LIN {X 0,Y 288.913,Z 1256.965,A -85,B 0,C 180,E1 22492.445,E2 22492.445} C_VEL
LIN {X 0,Y 288.678,Z 1266.037,A -85,B 0,C 180,E1 22499.979,E2 22499.979} C_VEL
LIN {X 0,Y 289.252,Z 1269.357,A -85,B 0,C 180,E1 22505.992,E2 22505.992} C_VEL
LIN {X 0,Y 291.406,Z 1269.606,A -85,B 0,C 180,E1 22511.982,E2 22511.982} C_VEL
LIN {X 0,Y 298.511,Z 1264.594,A -85,B 0,C 180,E1 22520.789,E2 22520.789} C_VEL
LIN {X 0,Y 311.662,Z 1253.252,A -85,B 0,C 180,E1 22529.064,E2 22529.064} C_VEL
LIN {X 0,Y 331.336,Z 1236.016,A -85,B 0,C 180,E1 22536.45,E2 22536.45} C_VEL
LIN {X 0,Y 358.772,Z 1211.951,A -85,B 0,C 180,E1 22542.947,E2 22542.947} C_VEL
LIN {X 0,Y 361.993,Z 1209.216,A -85,B 0,C 180,E1 22543.83,E2 22543.83} C_VEL
LIN {X 0,Y 333.812,Z 1237.362,A -85,B 0,C 180,E1 22549.712,E2 22549.712} C_VEL
LIN {X 0,Y 313.92,Z 1258.852,A -85,B 0,C 180,E1 22556.298,E2 22556.298} C_VEL
LIN {X 0,Y 299.966,Z 1275.518,A -85,B 0,C 180,E1 22563.783,E2 22563.783} C_VEL
LIN {X 0,Y 291.853,Z 1286.905,A -85,B 0,C 180,E1 22571.864,E2 22571.864} C_VEL
LIN {X 0,Y 289.278,Z 1291.684,A -85,B 0,C 180,E1 22577.92,E2 22577.92} C_VEL
LIN {X 0,Y 288.568,Z 1293.172,A -85,B 0,C 180,E1 22585.704,E2 22585.704} C_VEL
LIN {X 0,Y 288.992,Z 1290.468,A -85,B 0,C 180,E1 22591.516,E2 22591.516} C_VEL
LIN {X 0,Y 289.159,Z 1283.794,A -85,B 0,C 180,E1 22597.542,E2 22597.542} C_VEL
LIN {X 0,Y 290.047,Z 1270.937,A -85,B 0,C 180,E1 22604.382,E2 22604.382} C_VEL
LIN {X 0,Y 290.956,Z 1264.711,A -85,B 0,C 180,E1 22607.439,E2 22607.439} C_VEL
LIN {X 0,Y 296.193,Z 1251.831,A -85,B 0,C 180,E1 22614.979,E2 22614.979} C_VEL
LIN {X 0,Y 306.956,Z 1232.131,A -85,B 0,C 180,E1 22622.484,E2 22622.484} C_VEL
LIN {X 0,Y 322.234,Z 1206.9,A -85,B 0,C 180,E1 22628.957,E2 22628.957} C_VEL
LIN {X 0,Y 340.074,Z 1177.254,A -85,B 0,C 180,E1 22634.139,E2 22634.139} C_VEL
LIN {X 0,Y 358.674,Z 1143.561,A -85,B 0,C 180,E1 22638.141,E2 22638.141} C_VEL
LIN {X 0,Y 372.662,Z 1114.646,A -85,B 0,C 180,E1 22640.6,E2 22640.6} C_VEL
LIN {X 0,Y 373.421,Z 1108.193,A -85,B 0,C 180,E1 22642.533,E2 22642.533} C_VEL
LIN {X 0,Y 372.674,Z 1104.982,A -85,B 0,C 180,E1 22645.328,E2 22645.328} C_VEL
LIN {X 0,Y 372.153,Z 1105.867,A -85,B 0,C 180,E1 22648.785,E2 22648.785} C_VEL
LIN {X 0,Y 371.792,Z 1111.104,A -85,B 0,C 180,E1 22651.662,E2 22651.662} C_VEL
LIN {X 0,Y 356.868,Z 1141.073,A -85,B 0,C 180,E1 22654.392,E2 22654.392} C_VEL
LIN {X 0,Y 341.823,Z 1166.001,A -85,B 0,C 180,E1 22657.887,E2 22657.887} C_VEL
LIN {X 0,Y 327.191,Z 1186.173,A -85,B 0,C 180,E1 22662.219,E2 22662.219} C_VEL
LIN {X 0,Y 325.799,Z 1187.915,A -85,B 0,C 180,E1 22662.7,E2 22662.7} C_VEL
LIN {X 0,Y 316.07,Z 1196.775,A -85,B 0,C 180,E1 22664.784,E2 22664.784} C_VEL
LIN {X 0,Y 307.469,Z 1203.336,A -85,B 0,C 180,E1 22666.77,E2 22666.77} C_VEL
LIN {X 0,Y 306.628,Z 1204.067,A -85,B 0,C 180,E1 22667.118,E2 22667.118} C_VEL
LIN {X 0,Y 296.611,Z 1212.121,A -85,B 0,C 180,E1 22672.684,E2 22672.684} C_VEL
LIN {X 0,Y 291.006,Z 1214.857,A -85,B 0,C 180,E1 22677.037,E2 22677.037} C_VEL
LIN {X 0,Y 285.807,Z 1214.307,A -85,B 0,C 180,E1 22683.06,E2 22683.06} C_VEL
LIN {X 0,Y 283.385,Z 1208.666,A -85,B 0,C 180,E1 22689.252,E2 22689.252} C_VEL
LIN {X 0,Y 283.421,Z 1196.875,A -85,B 0,C 180,E1 22695.723,E2 22695.723} C_VEL
LIN {X 0,Y 285.142,Z 1180.307,A -85,B 0,C 180,E1 22701.438,E2 22701.438} C_VEL
LIN {X 0,Y 288.35,Z 1157.172,A -85,B 0,C 180,E1 22706.829,E2 22706.829} C_VEL
LIN {X 0,Y 292.258,Z 1130.682,A -85,B 0,C 180,E1 22711.033,E2 22711.033} C_VEL
LIN {X 0,Y 296.178,Z 1100.104,A -85,B 0,C 180,E1 22714.268,E2 22714.268} C_VEL
LIN {X 0,Y 299.485,Z 1062.201,A -85,B 0,C 180,E1 22716.707,E2 22716.707} C_VEL
LIN {X 0,Y 298.982,Z 1051.383,A -85,B 0,C 180,E1 22717.371,E2 22717.371} C_VEL
LIN {X 0,Y 282.969,Z 995.061,A -85,B 0,C 180,E1 22721.869,E2 22721.869} C_VEL
LIN {X 0,Y 277.408,Z 977.53,A -85,B 0,C 180,E1 22723.544,E2 22723.544} C_VEL
LIN {X 0,Y 277.257,Z 977.53,A -85,B 0,C 180,E1 22733.028,E2 22733.028} C_VEL
LIN {X 0,Y 277.681,Z 977.53,A -85,B 0,C 180,E1 22740.854,E2 22740.854} C_VEL
LIN {X 0,Y 278.202,Z 977.53,A -85,B 0,C 180,E1 22747.851,E2 22747.851} C_VEL
LIN {X 0,Y 278.682,Z 977.53,A -85,B 0,C 180,E1 22754.21,E2 22754.21} C_VEL
LIN {X 0,Y 279.215,Z 977.53,A -85,B 0,C 180,E1 22760.616,E2 22760.616} C_VEL
LIN {X 0,Y 279.937,Z 977.53,A -85,B 0,C 180,E1 22766.883,E2 22766.883} C_VEL
LIN {X 0,Y 279.933,Z 977.53,A -85,B 0,C 180,E1 22773.088,E2 22773.088} C_VEL
LIN {X 0,Y 278.942,Z 977.53,A -85,B 0,C 180,E1 22782.535,E2 22782.535} C_VEL
LIN {X 0,Y 278.361,Z 977.53,A -85,B 0,C 180,E1 22789.048,E2 22789.048} C_VEL
LIN {X 0,Y 277.861,Z 977.53,A -85,B 0,C 180,E1 22795.85,E2 22795.85} C_VEL
LIN {X 0,Y 277.467,Z 977.53,A -85,B 0,C 180,E1 22804.97,E2 22804.97} C_VEL
LIN {X 0,Y 277.579,Z 977.96,A -85,B 0,C 180,E1 22805.92,E2 22805.92} C_VEL
LIN {X 0,Y 300.397,Z 1034.729,A -85,B 0,C 180,E1 22811.695,E2 22811.695} C_VEL
LIN {X 0,Y 313.014,Z 1073.998,A -85,B 0,C 180,E1 22815.793,E2 22815.793} C_VEL
LIN {X 0,Y 317.958,Z 1093.026,A -85,B 0,C 180,E1 22817.944,E2 22817.944} C_VEL
LIN {X 0,Y 309.265,Z 1133.148,A -85,B 0,C 180,E1 22821.776,E2 22821.776} C_VEL
LIN {X 0,Y 300.222,Z 1169.342,A -85,B 0,C 180,E1 22826.69,E2 22826.69} C_VEL
LIN {X 0,Y 292.592,Z 1198.797,A -85,B 0,C 180,E1 22832.199,E2 22832.199} C_VEL
LIN {X 0,Y 286.541,Z 1224.077,A -85,B 0,C 180,E1 22838.661,E2 22838.661} C_VEL
LIN {X 0,Y 282.581,Z 1244.505,A -85,B 0,C 180,E1 22846.016,E2 22846.016} C_VEL
LIN {X 0,Y 280.968,Z 1257.783,A -85,B 0,C 180,E1 22853.009,E2 22853.009} C_VEL
LIN {X 0,Y 280.777,Z 1266.014,A -85,B 0,C 180,E1 22859.978,E2 22859.978} C_VEL
LIN {X 0,Y 281.383,Z 1269.716,A -85,B 0,C 180,E1 22866.16,E2 22866.16} C_VEL
LIN {X 0,Y 283.679,Z 1270.268,A -85,B 0,C 180,E1 22872.313,E2 22872.313} C_VEL
LIN {X 0,Y 291.207,Z 1265.806,A -85,B 0,C 180,E1 22881.335,E2 22881.335} C_VEL
LIN {X 0,Y 305.036,Z 1255.326,A -85,B 0,C 180,E1 22889.758,E2 22889.758} C_VEL
LIN {X 0,Y 327.34,Z 1237.562,A -85,B 0,C 180,E1 22897.738,E2 22897.738} C_VEL
LIN {X 0,Y 352.425,Z 1217.519,A -85,B 0,C 180,E1 22903.435,E2 22903.435} C_VEL
LIN {X 0,Y 349.967,Z 1219.814,A -85,B 0,C 180,E1 22904.214,E2 22904.214} C_VEL
LIN {X 0,Y 319.893,Z 1247.945,A -85,B 0,C 180,E1 22911.141,E2 22911.141} C_VEL
LIN {X 0,Y 298.473,Z 1269.792,A -85,B 0,C 180,E1 22919.607,E2 22919.607} C_VEL
LIN {X 0,Y 286.72,Z 1283.669,A -85,B 0,C 180,E1 22928.303,E2 22928.303} C_VEL
LIN {X 0,Y 282.382,Z 1289.896,A -85,B 0,C 180,E1 22934.881,E2 22934.881} C_VEL
LIN {X 0,Y 280.916,Z 1292.547,A -85,B 0,C 180,E1 22940.702,E2 22940.702} C_VEL
LIN {X 0,Y 280.835,Z 1292.257,A -85,B 0,C 180,E1 22946.921,E2 22946.921} C_VEL
LIN {X 0,Y 281.131,Z 1289.623,A -85,B 0,C 180,E1 22951.559,E2 22951.559} C_VEL
LIN {X 0,Y 281.302,Z 1282.585,A -85,B 0,C 180,E1 22957.754,E2 22957.754} C_VEL
LIN {X 0,Y 282.209,Z 1270.064,A -85,B 0,C 180,E1 22964.483,E2 22964.483} C_VEL
LIN {X 0,Y 282.953,Z 1265.098,A -85,B 0,C 180,E1 22967.145,E2 22967.145} C_VEL
LIN {X 0,Y 288.891,Z 1251.656,A -85,B 0,C 180,E1 22975.656,E2 22975.656} C_VEL
LIN {X 0,Y 300.247,Z 1232.56,A -85,B 0,C 180,E1 22983.303,E2 22983.303} C_VEL
LIN {X 0,Y 316.069,Z 1208.342,A -85,B 0,C 180,E1 22989.806,E2 22989.806} C_VEL
LIN {X 0,Y 334.659,Z 1179.668,A -85,B 0,C 180,E1 22995.033,E2 22995.033} C_VEL
LIN {X 0,Y 353.859,Z 1147.347,A -85,B 0,C 180,E1 22999.018,E2 22999.018} C_VEL
LIN {X 0,Y 368.467,Z 1119.396,A -85,B 0,C 180,E1 23001.401,E2 23001.401} C_VEL
LIN {X 0,Y 369.311,Z 1113.908,A -85,B 0,C 180,E1 23003.254,E2 23003.254} C_VEL
LIN {X 0,Y 368.846,Z 1111.925,A -85,B 0,C 180,E1 23005.267,E2 23005.267} C_VEL
LIN {X 0,Y 368.267,Z 1112.965,A -85,B 0,C 180,E1 23008.847,E2 23008.847} C_VEL
LIN {X 0,Y 368.026,Z 1115.337,A -85,B 0,C 180,E1 23010.415,E2 23010.415} C_VEL
LIN {X 0,Y 366.347,Z 1119.287,A -85,B 0,C 180,E1 23011.013,E2 23011.013} C_VEL
LIN {X 0,Y 350.419,Z 1148.17,A -85,B 0,C 180,E1 23013.886,E2 23013.886} C_VEL
LIN {X 0,Y 333.991,Z 1172.642,A -85,B 0,C 180,E1 23017.692,E2 23017.692} C_VEL
LIN {X 0,Y 318.539,Z 1191.796,A -85,B 0,C 180,E1 23022.323,E2 23022.323} C_VEL
LIN {X 0,Y 306.628,Z 1204.067,A -85,B 0,C 180,E1 23027.118,E2 23027.118} C_VEL
LIN {X 0,Y 297.424,Z 1209.949,A -85,B 0,C 180,E1 23029.73,E2 23029.73} C_VEL
LIN {X 0,Y 289.436,Z 1213.784,A -85,B 0,C 180,E1 23032.173,E2 23032.173} C_VEL
LIN {X 0,Y 288.735,Z 1214.113,A -85,B 0,C 180,E1 23032.578,E2 23032.578} C_VEL
LIN {X 0,Y 283.133,Z 1216.283,A -85,B 0,C 180,E1 23036.954,E2 23036.954} C_VEL
LIN {X 0,Y 277.875,Z 1215.064,A -85,B 0,C 180,E1 23043.148,E2 23043.148} C_VEL
LIN {X 0,Y 275.444,Z 1208.736,A -85,B 0,C 180,E1 23049.521,E2 23049.521} C_VEL
LIN {X 0,Y 275.571,Z 1196.71,A -85,B 0,C 180,E1 23055.979,E2 23055.979} C_VEL
LIN {X 0,Y 277.478,Z 1179.1,A -85,B 0,C 180,E1 23061.994,E2 23061.994} C_VEL
LIN {X 0,Y 280.65,Z 1156.661,A -85,B 0,C 180,E1 23067.205,E2 23067.205} C_VEL
LIN {X 0,Y 284.652,Z 1130.227,A -85,B 0,C 180,E1 23071.456,E2 23071.456} C_VEL
LIN {X 0,Y 288.634,Z 1099.807,A -85,B 0,C 180,E1 23074.721,E2 23074.721} C_VEL
LIN {X 0,Y 292.247,Z 1059.09,A -85,B 0,C 180,E1 23077.358,E2 23077.358} C_VEL
LIN {X 0,Y 281.853,Z 1016.879,A -85,B 0,C 180,E1 23080.687,E2 23080.687} C_VEL
LIN {X 0,Y 269.397,Z 977.53,A -85,B 0,C 180,E1 23084.328,E2 23084.328} C_VEL
LIN {X 0,Y 269.242,Z 977.53,A -85,B 0,C 180,E1 23092.019,E2 23092.019} C_VEL
LIN {X 0,Y 269.549,Z 977.53,A -85,B 0,C 180,E1 23099.589,E2 23099.589} C_VEL
LIN {X 0,Y 270.123,Z 977.53,A -85,B 0,C 180,E1 23106.863,E2 23106.863} C_VEL
LIN {X 0,Y 270.679,Z 977.53,A -85,B 0,C 180,E1 23113.73,E2 23113.73} C_VEL
LIN {X 0,Y 271.289,Z 977.53,A -85,B 0,C 180,E1 23120.339,E2 23120.339} C_VEL
LIN {X 0,Y 272.024,Z 977.53,A -85,B 0,C 180,E1 23126.792,E2 23126.792} C_VEL
LIN {X 0,Y 272.019,Z 977.53,A -85,B 0,C 180,E1 23133.178,E2 23133.178} C_VEL
LIN {X 0,Y 271.263,Z 977.53,A -85,B 0,C 180,E1 23139.632,E2 23139.632} C_VEL
LIN {X 0,Y 270.47,Z 977.53,A -85,B 0,C 180,E1 23147.696,E2 23147.696} C_VEL
LIN {X 0,Y 269.94,Z 977.53,A -85,B 0,C 180,E1 23156.048,E2 23156.048} C_VEL
LIN {X 0,Y 269.572,Z 977.695,A -85,B 0,C 180,E1 23164.793,E2 23164.793} C_VEL
LIN {X 0,Y 292.525,Z 1034.518,A -85,B 0,C 180,E1 23170.823,E2 23170.823} C_VEL
LIN {X 0,Y 305.526,Z 1075.222,A -85,B 0,C 180,E1 23175.204,E2 23175.204} C_VEL
LIN {X 0,Y 310.377,Z 1095.235,A -85,B 0,C 180,E1 23177.517,E2 23177.517} C_VEL
LIN {X 0,Y 301.699,Z 1134.071,A -85,B 0,C 180,E1 23181.347,E2 23181.347} C_VEL
LIN {X 0,Y 292.601,Z 1169.644,A -85,B 0,C 180,E1 23186.3,E2 23186.3} C_VEL
LIN {X 0,Y 284.518,Z 1200.304,A -85,B 0,C 180,E1 23192.204,E2 23192.204} C_VEL
LIN {X 0,Y 278.158,Z 1226.524,A -85,B 0,C 180,E1 23199.241,E2 23199.241} C_VEL
LIN {X 0,Y 274.526,Z 1245.536,A -85,B 0,C 180,E1 23206.448,E2 23206.448} C_VEL
LIN {X 0,Y 273.004,Z 1258.55,A -85,B 0,C 180,E1 23213.605,E2 23213.605} C_VEL
LIN {X 0,Y 272.903,Z 1265.954,A -85,B 0,C 180,E1 23219.977,E2 23219.977} C_VEL
LIN {X 0,Y 273.53,Z 1270.023,A -85,B 0,C 180,E1 23226.337,E2 23226.337} C_VEL
LIN {X 0,Y 275.96,Z 1270.937,A -85,B 0,C 180,E1 23232.663,E2 23232.663} C_VEL
LIN {X 0,Y 283.929,Z 1267.034,A -85,B 0,C 180,E1 23241.91,E2 23241.91} C_VEL
LIN {X 0,Y 298.433,Z 1257.296,A -85,B 0,C 180,E1 23250.485,E2 23250.485} C_VEL
LIN {X 0,Y 321.645,Z 1240.685,A -85,B 0,C 180,E1 23258.527,E2 23258.527} C_VEL
LIN {X 0,Y 342.424,Z 1225.545,A -85,B 0,C 180,E1 23263.266,E2 23263.266} C_VEL
LIN {X 0,Y 343.123,Z 1225.113,A -85,B 0,C 180,E1 23263.689,E2 23263.689} C_VEL
LIN {X 0,Y 312.004,Z 1251.858,A -85,B 0,C 180,E1 23270.867,E2 23270.867} C_VEL
LIN {X 0,Y 289.855,Z 1272.711,A -85,B 0,C 180,E1 23279.817,E2 23279.817} C_VEL
LIN {X 0,Y 277.869,Z 1285.614,A -85,B 0,C 180,E1 23289.256,E2 23289.256} C_VEL
LIN {X 0,Y 273.627,Z 1291.227,A -85,B 0,C 180,E1 23297.218,E2 23297.218} C_VEL
LIN {X 0,Y 272.852,Z 1292.257,A -85,B 0,C 180,E1 23303.638,E2 23303.638} C_VEL
LIN {X 0,Y 273.451,Z 1289.888,A -85,B 0,C 180,E1 23310.015,E2 23310.015} C_VEL
LIN {X 0,Y 273.431,Z 1282.535,A -85,B 0,C 180,E1 23317.178,E2 23317.178} C_VEL
LIN {X 0,Y 274.227,Z 1270.393,A -85,B 0,C 180,E1 23324.035,E2 23324.035} C_VEL
LIN {X 0,Y 274.729,Z 1266.131,A -85,B 0,C 180,E1 23326.023,E2 23326.023} C_VEL
LIN {X 0,Y 279.954,Z 1254.348,A -85,B 0,C 180,E1 23334.817,E2 23334.817} C_VEL
LIN {X 0,Y 291.472,Z 1236.104,A -85,B 0,C 180,E1 23343.1,E2 23343.1} C_VEL
LIN {X 0,Y 308.83,Z 1211.57,A -85,B 0,C 180,E1 23350.288,E2 23350.288} C_VEL
LIN {X 0,Y 327.127,Z 1185.458,A -85,B 0,C 180,E1 23355.43,E2 23355.43} C_VEL
LIN {X 0,Y 347.783,Z 1153.343,A -85,B 0,C 180,E1 23359.7,E2 23359.7} C_VEL
LIN {X 0,Y 364.712,Z 1123.183,A -85,B 0,C 180,E1 23362.414,E2 23362.414} C_VEL
LIN {X 0,Y 364.999,Z 1119.391,A -85,B 0,C 180,E1 23364.491,E2 23364.491} C_VEL
LIN {X 0,Y 364.303,Z 1119.747,A -85,B 0,C 180,E1 23368.697,E2 23368.697} C_VEL
LIN {X 0,Y 364.038,Z 1121.221,A -85,B 0,C 180,E1 23369.767,E2 23369.767} C_VEL
LIN {X 0,Y 345.85,Z 1151.99,A -85,B 0,C 180,E1 23372.987,E2 23372.987} C_VEL
LIN {X 0,Y 329.86,Z 1174.28,A -85,B 0,C 180,E1 23376.537,E2 23376.537} C_VEL
LIN {X 0,Y 314.161,Z 1192.55,A -85,B 0,C 180,E1 23380.978,E2 23380.978} C_VEL
LIN {X 0,Y 299.904,Z 1206.191,A -85,B 0,C 180,E1 23386.447,E2 23386.447} C_VEL
LIN {X 0,Y 288.735,Z 1214.113,A -85,B 0,C 180,E1 23392.578,E2 23392.578} C_VEL
LIN {X 0,Y 280.597,Z 1216.672,A -85,B 0,C 180,E1 23395.659,E2 23395.659} C_VEL
LIN {X 0,Y 273.689,Z 1217.548,A -85,B 0,C 180,E1 23398.479,E2 23398.479} C_VEL
LIN {X 0,Y 273.183,Z 1217.478,A -85,B 0,C 180,E1 23398.924,E2 23398.924} C_VEL
LIN {X 0,Y 269.062,Z 1214.432,A -85,B 0,C 180,E1 23404.868,E2 23404.868} C_VEL
LIN {X 0,Y 267.38,Z 1206.14,A -85,B 0,C 180,E1 23411.463,E2 23411.463} C_VEL
LIN {X 0,Y 268.135,Z 1191.668,A -85,B 0,C 180,E1 23418.13,E2 23418.13} C_VEL
LIN {X 0,Y 270.499,Z 1172.473,A -85,B 0,C 180,E1 23423.984,E2 23423.984} C_VEL
LIN {X 0,Y 274.256,Z 1148.078,A -85,B 0,C 180,E1 23429.086,E2 23429.086} C_VEL
LIN {X 0,Y 278.482,Z 1119.043,A -85,B 0,C 180,E1 23433.219,E2 23433.219} C_VEL
LIN {X 0,Y 282.397,Z 1086.606,A -85,B 0,C 180,E1 23436.195,E2 23436.195} C_VEL
LIN {X 0,Y 284.42,Z 1056.353,A -85,B 0,C 180,E1 23438.064,E2 23438.064} C_VEL
LIN {X 0,Y 269.303,Z 1001.916,A -85,B 0,C 180,E1 23442.706,E2 23442.706} C_VEL
LIN {X 0,Y 261.427,Z 977.53,A -85,B 0,C 180,E1 23445.044,E2 23445.044} C_VEL
LIN {X 0,Y 261.299,Z 977.53,A -85,B 0,C 180,E1 23454.538,E2 23454.538} C_VEL
LIN {X 0,Y 261.789,Z 977.53,A -85,B 0,C 180,E1 23462.399,E2 23462.399} C_VEL
LIN {X 0,Y 262.369,Z 977.53,A -85,B 0,C 180,E1 23469.709,E2 23469.709} C_VEL
LIN {X 0,Y 263.089,Z 977.53,A -85,B 0,C 180,E1 23478.353,E2 23478.353} C_VEL
LIN {X 0,Y 264.09,Z 977.53,A -85,B 0,C 180,E1 23486.695,E2 23486.695} C_VEL
LIN {X 0,Y 264.478,Z 977.53,A -85,B 0,C 180,E1 23489.985,E2 23489.985} C_VEL
LIN {X 0,Y 263.652,Z 977.53,A -85,B 0,C 180,E1 23496.585,E2 23496.585} C_VEL
LIN {X 0,Y 262.984,Z 977.53,A -85,B 0,C 180,E1 23503.309,E2 23503.309} C_VEL
LIN {X 0,Y 262.183,Z 977.53,A -85,B 0,C 180,E1 23512.331,E2 23512.331} C_VEL
LIN {X 0,Y 261.6,Z 977.53,A -85,B 0,C 180,E1 23521.402,E2 23521.402} C_VEL
LIN {X 0,Y 261.605,Z 977.53,A -85,B 0,C 180,E1 23523.583,E2 23523.583} C_VEL
LIN {X 0,Y 284.39,Z 1033.772,A -85,B 0,C 180,E1 23529.851,E2 23529.851} C_VEL
LIN {X 0,Y 297.241,Z 1073.785,A -85,B 0,C 180,E1 23534.297,E2 23534.297} C_VEL
LIN {X 0,Y 302.876,Z 1096.857,A -85,B 0,C 180,E1 23537.031,E2 23537.031} C_VEL
LIN {X 0,Y 293.687,Z 1136.512,A -85,B 0,C 180,E1 23541.092,E2 23541.092} C_VEL
LIN {X 0,Y 284.47,Z 1171.588,A -85,B 0,C 180,E1 23546.175,E2 23546.175} C_VEL
LIN {X 0,Y 276.388,Z 1201.702,A -85,B 0,C 180,E1 23552.203,E2 23552.203} C_VEL
LIN {X 0,Y 270.331,Z 1226.439,A -85,B 0,C 180,E1 23559.042,E2 23559.042} C_VEL
LIN {X 0,Y 266.477,Z 1246.367,A -85,B 0,C 180,E1 23566.831,E2 23566.831} C_VEL
LIN {X 0,Y 265.029,Z 1259.283,A -85,B 0,C 180,E1 23574.235,E2 23574.235} C_VEL
LIN {X 0,Y 265,Z 1267.449,A -85,B 0,C 180,E1 23581.779,E2 23581.779} C_VEL
LIN {X 0,Y 266.684,Z 1271.263,A -85,B 0,C 180,E1 23589.79,E2 23589.79} C_VEL
LIN {X 0,Y 273.176,Z 1270.019,A -85,B 0,C 180,E1 23599.49,E2 23599.49} C_VEL
LIN {X 0,Y 286.075,Z 1262.888,A -85,B 0,C 180,E1 23608.442,E2 23608.442} C_VEL
LIN {X 0,Y 307.827,Z 1249.109,A -85,B 0,C 180,E1 23617.055,E2 23617.055} C_VEL
LIN {X 0,Y 334.212,Z 1231.755,A -85,B 0,C 180,E1 23623.514,E2 23623.514} C_VEL
LIN {X 0,Y 302.811,Z 1256.641,A -85,B 0,C 180,E1 23630.98,E2 23630.98} C_VEL
LIN {X 0,Y 281.712,Z 1274.755,A -85,B 0,C 180,E1 23639.735,E2 23639.735} C_VEL
LIN {X 0,Y 270.386,Z 1285.758,A -85,B 0,C 180,E1 23648.654,E2 23648.654} C_VEL
LIN {X 0,Y 265.814,Z 1290.899,A -85,B 0,C 180,E1 23656.835,E2 23656.835} C_VEL
LIN {X 0,Y 264.965,Z 1291.615,A -85,B 0,C 180,E1 23663.448,E2 23663.448} C_VEL
LIN {X 0,Y 265.59,Z 1289.004,A -85,B 0,C 180,E1 23670.015,E2 23670.015} C_VEL
LIN {X 0,Y 265.618,Z 1282.453,A -85,B 0,C 180,E1 23676.567,E2 23676.567} C_VEL
LIN {X 0,Y 266.388,Z 1269.417,A -85,B 0,C 180,E1 23684.14,E2 23684.14} C_VEL
LIN {X 0,Y 266.951,Z 1265.43,A -85,B 0,C 180,E1 23686.503,E2 23686.503} C_VEL
LIN {X 0,Y 272.632,Z 1254.122,A -85,B 0,C 180,E1 23695.531,E2 23695.531} C_VEL
LIN {X 0,Y 284.723,Z 1236.648,A -85,B 0,C 180,E1 23703.928,E2 23703.928} C_VEL
LIN {X 0,Y 303.208,Z 1212.52,A -85,B 0,C 180,E1 23711.336,E2 23711.336} C_VEL
LIN {X 0,Y 323.05,Z 1186.132,A -85,B 0,C 180,E1 23716.656,E2 23716.656} C_VEL
LIN {X 0,Y 344.466,Z 1155.025,A -85,B 0,C 180,E1 23720.851,E2 23720.851} C_VEL
LIN {X 0,Y 360.571,Z 1128.224,A -85,B 0,C 180,E1 23723.279,E2 23723.279} C_VEL
LIN {X 0,Y 360.841,Z 1126.758,A -85,B 0,C 180,E1 23724.018,E2 23724.018} C_VEL
LIN {X 0,Y 360.377,Z 1125.639,A -85,B 0,C 180,E1 23727.259,E2 23727.259} C_VEL
LIN {X 0,Y 360.15,Z 1126.687,A -85,B 0,C 180,E1 23728.72,E2 23728.72} C_VEL
LIN {X 0,Y 358.204,Z 1130.191,A -85,B 0,C 180,E1 23729.273,E2 23729.273} C_VEL
LIN {X 0,Y 340.77,Z 1156.86,A -85,B 0,C 180,E1 23732.19,E2 23732.19} C_VEL
LIN {X 0,Y 323.148,Z 1179.267,A -85,B 0,C 180,E1 23736.02,E2 23736.02} C_VEL
LIN {X 0,Y 304.998,Z 1198.25,A -85,B 0,C 180,E1 23741.186,E2 23741.186} C_VEL
LIN {X 0,Y 290.118,Z 1210.593,A -85,B 0,C 180,E1 23747.198,E2 23747.198} C_VEL
LIN {X 0,Y 279.005,Z 1216.753,A -85,B 0,C 180,E1 23753.787,E2 23753.787} C_VEL
LIN {X 0,Y 273.183,Z 1217.478,A -85,B 0,C 180,E1 23758.924,E2 23758.924} C_VEL
LIN {X 0,Y 266.523,Z 1216.607,A -85,B 0,C 180,E1 23762.364,E2 23762.364} C_VEL
LIN {X 0,Y 260.699,Z 1213.899,A -85,B 0,C 180,E1 23765.916,E2 23765.916} C_VEL
LIN {X 0,Y 259.482,Z 1204.285,A -85,B 0,C 180,E1 23772.672,E2 23772.672} C_VEL
LIN {X 0,Y 260.557,Z 1189.4,A -85,B 0,C 180,E1 23779.117,E2 23779.117} C_VEL
LIN {X 0,Y 263.226,Z 1168.701,A -85,B 0,C 180,E1 23785.145,E2 23785.145} C_VEL
LIN {X 0,Y 267.397,Z 1143.375,A -85,B 0,C 180,E1 23790.216,E2 23790.216} C_VEL
LIN {X 0,Y 271.543,Z 1114.089,A -85,B 0,C 180,E1 23794.183,E2 23794.183} C_VEL
LIN {X 0,Y 275.19,Z 1082.564,A -85,B 0,C 180,E1 23796.931,E2 23796.931} C_VEL
LIN {X 0,Y 276.819,Z 1057.583,A -85,B 0,C 180,E1 23798.525,E2 23798.525} C_VEL
LIN {X 0,Y 261.766,Z 1003.117,A -85,B 0,C 180,E1 23803.348,E2 23803.348} C_VEL
LIN {X 0,Y 253.452,Z 977.53,A -85,B 0,C 180,E1 23805.993,E2 23805.993} C_VEL
LIN {X 0,Y 253.231,Z 977.53,A -85,B 0,C 180,E1 23813.227,E2 23813.227} C_VEL
LIN {X 0,Y 253.771,Z 977.53,A -85,B 0,C 180,E1 23821.448,E2 23821.448} C_VEL
LIN {X 0,Y 254.402,Z 977.53,A -85,B 0,C 180,E1 23829.044,E2 23829.044} C_VEL
LIN {X 0,Y 254.993,Z 977.53,A -85,B 0,C 180,E1 23836.233,E2 23836.233} C_VEL
LIN {X 0,Y 255.718,Z 977.53,A -85,B 0,C 180,E1 23843.178,E2 23843.178} C_VEL
LIN {X 0,Y 256.567,Z 977.53,A -85,B 0,C 180,E1 23849.984,E2 23849.984} C_VEL
LIN {X 0,Y 255.695,Z 977.53,A -85,B 0,C 180,E1 23856.791,E2 23856.791} C_VEL
LIN {X 0,Y 254.987,Z 977.53,A -85,B 0,C 180,E1 23863.735,E2 23863.735} C_VEL
LIN {X 0,Y 254.371,Z 977.53,A -85,B 0,C 180,E1 23870.924,E2 23870.924} C_VEL
LIN {X 0,Y 253.696,Z 977.53,A -85,B 0,C 180,E1 23880.692,E2 23880.692} C_VEL
LIN {X 0,Y 253.665,Z 977.557,A -85,B 0,C 180,E1 23882.388,E2 23882.388} C_VEL
LIN {X 0,Y 276.536,Z 1033.578,A -85,B 0,C 180,E1 23888.915,E2 23888.915} C_VEL
LIN {X 0,Y 289.461,Z 1073.762,A -85,B 0,C 180,E1 23893.523,E2 23893.523} C_VEL
LIN {X 0,Y 295.553,Z 1097.709,A -85,B 0,C 180,E1 23896.472,E2 23896.472} C_VEL
LIN {X 0,Y 285.937,Z 1138.05,A -85,B 0,C 180,E1 23900.735,E2 23900.735} C_VEL
LIN {X 0,Y 276.703,Z 1172.33,A -85,B 0,C 180,E1 23905.848,E2 23905.848} C_VEL
LIN {X 0,Y 268.256,Z 1203.166,A -85,B 0,C 180,E1 23912.235,E2 23912.235} C_VEL
LIN {X 0,Y 261.926,Z 1228.693,A -85,B 0,C 180,E1 23919.667,E2 23919.667} C_VEL
LIN {X 0,Y 258.445,Z 1247.235,A -85,B 0,C 180,E1 23927.276,E2 23927.276} C_VEL
LIN {X 0,Y 257.075,Z 1259.988,A -85,B 0,C 180,E1 23934.904,E2 23934.904} C_VEL
LIN {X 0,Y 257.112,Z 1267.219,A -85,B 0,C 180,E1 23941.664,E2 23941.664} C_VEL
LIN {X 0,Y 258.895,Z 1271.615,A -85,B 0,C 180,E1 23950.087,E2 23950.087} C_VEL
LIN {X 0,Y 265.679,Z 1271.021,A -85,B 0,C 180,E1 23959.984,E2 23959.984} C_VEL
LIN {X 0,Y 279.318,Z 1264.646,A -85,B 0,C 180,E1 23969.196,E2 23969.196} C_VEL
LIN {X 0,Y 301.933,Z 1251.806,A -85,B 0,C 180,E1 23977.904,E2 23977.904} C_VEL
LIN {X 0,Y 322.487,Z 1239.601,A -85,B 0,C 180,E1 23982.995,E2 23982.995} C_VEL
LIN {X 0,Y 323.735,Z 1238.967,A -85,B 0,C 180,E1 23983.618,E2 23983.618} C_VEL
LIN {X 0,Y 294.309,Z 1260.485,A -85,B 0,C 180,E1 23990.863,E2 23990.863} C_VEL
LIN {X 0,Y 272.956,Z 1277.216,A -85,B 0,C 180,E1 24000.042,E2 24000.042} C_VEL
LIN {X 0,Y 261.527,Z 1287.172,A -85,B 0,C 180,E1 24009.674,E2 24009.674} C_VEL
LIN {X 0,Y 257.31,Z 1291.142,A -85,B 0,C 180,E1 24019.84,E2 24019.84} C_VEL
LIN {X 0,Y 257.234,Z 1289.968,A -85,B 0,C 180,E1 24026.639,E2 24026.639} C_VEL
LIN {X 0,Y 257.593,Z 1286.56,A -85,B 0,C 180,E1 24031.87,E2 24031.87} C_VEL
LIN {X 0,Y 257.784,Z 1278.791,A -85,B 0,C 180,E1 24038.466,E2 24038.466} C_VEL
LIN {X 0,Y 258.891,Z 1265.808,A -85,B 0,C 180,E1 24045.566,E2 24045.566} C_VEL
LIN {X 0,Y 263.703,Z 1256.288,A -85,B 0,C 180,E1 24054.636,E2 24054.636} C_VEL
LIN {X 0,Y 275.363,Z 1240.507,A -85,B 0,C 180,E1 24063.404,E2 24063.404} C_VEL
LIN {X 0,Y 293.752,Z 1218.294,A -85,B 0,C 180,E1 24071.142,E2 24071.142} C_VEL
LIN {X 0,Y 315.482,Z 1191.694,A -85,B 0,C 180,E1 24077.112,E2 24077.112} C_VEL
LIN {X 0,Y 338.549,Z 1160.884,A -85,B 0,C 180,E1 24081.579,E2 24081.579} C_VEL
LIN {X 0,Y 355.597,Z 1134.886,A -85,B 0,C 180,E1 24084.078,E2 24084.078} C_VEL
LIN {X 0,Y 356.413,Z 1133.202,A -85,B 0,C 180,E1 24084.483,E2 24084.483} C_VEL
LIN {X 0,Y 356.035,Z 1132.551,A -85,B 0,C 180,E1 24087.589,E2 24087.589} C_VEL
LIN {X 0,Y 355.259,Z 1133.956,A -85,B 0,C 180,E1 24088.24,E2 24088.24} C_VEL
LIN {X 0,Y 335.734,Z 1161.55,A -85,B 0,C 180,E1 24091.37,E2 24091.37} C_VEL
LIN {X 0,Y 316.659,Z 1183.874,A -85,B 0,C 180,E1 24095.423,E2 24095.423} C_VEL
LIN {X 0,Y 297.892,Z 1201.737,A -85,B 0,C 180,E1 24100.719,E2 24100.719} C_VEL
LIN {X 0,Y 284.114,Z 1212.101,A -85,B 0,C 180,E1 24106.138,E2 24106.138} C_VEL
LIN {X 0,Y 275.789,Z 1216.714,A -85,B 0,C 180,E1 24110.537,E2 24110.537} C_VEL
LIN {X 0,Y 267.352,Z 1218.852,A -85,B 0,C 180,E1 24116.775,E2 24116.775} C_VEL
LIN {X 0,Y 261.94,Z 1216.252,A -85,B 0,C 180,E1 24123.34,E2 24123.34} C_VEL
LIN {X 0,Y 260.699,Z 1213.899,A -85,B 0,C 180,E1 24125.916,E2 24125.916} C_VEL
LIN {X 0,Y 255.76,Z 1209.599,A -85,B 0,C 180,E1 24129.526,E2 24129.526} C_VEL
LIN {X 0,Y 251.6,Z 1203.635,A -85,B 0,C 180,E1 24133.142,E2 24133.142} C_VEL
LIN {X 0,Y 252.793,Z 1188.137,A -85,B 0,C 180,E1 24139.728,E2 24139.728} C_VEL
LIN {X 0,Y 255.67,Z 1166.843,A -85,B 0,C 180,E1 24145.844,E2 24145.844} C_VEL
LIN {X 0,Y 259.93,Z 1141.045,A -85,B 0,C 180,E1 24150.936,E2 24150.936} C_VEL
LIN {X 0,Y 264.169,Z 1112.66,A -85,B 0,C 180,E1 24154.773,E2 24154.773} C_VEL
LIN {X 0,Y 267.901,Z 1080.082,A -85,B 0,C 180,E1 24157.584,E2 24157.584} C_VEL
LIN {X 0,Y 269.124,Z 1058.526,A -85,B 0,C 180,E1 24159.013,E2 24159.013} C_VEL
LIN {X 0,Y 254.556,Z 1005.246,A -85,B 0,C 180,E1 24163.932,E2 24163.932} C_VEL
LIN {X 0,Y 245.435,Z 977.53,A -85,B 0,C 180,E1 24166.831,E2 24166.831} C_VEL
LIN {X 0,Y 245.393,Z 977.53,A -85,B 0,C 180,E1 24176.219,E2 24176.219} C_VEL
LIN {X 0,Y 246.041,Z 977.53,A -85,B 0,C 180,E1 24184.444,E2 24184.444} C_VEL
LIN {X 0,Y 246.697,Z 977.53,A -85,B 0,C 180,E1 24192.098,E2 24192.098} C_VEL
LIN {X 0,Y 247.38,Z 977.53,A -85,B 0,C 180,E1 24199.395,E2 24199.395} C_VEL
LIN {X 0,Y 248.237,Z 977.53,A -85,B 0,C 180,E1 24206.484,E2 24206.484} C_VEL
LIN {X 0,Y 248.656,Z 977.53,A -85,B 0,C 180,E1 24209.984,E2 24209.984} C_VEL
LIN {X 0,Y 247.737,Z 977.53,A -85,B 0,C 180,E1 24217.01,E2 24217.01} C_VEL
LIN {X 0,Y 246.989,Z 977.53,A -85,B 0,C 180,E1 24224.188,E2 24224.188} C_VEL
LIN {X 0,Y 246.218,Z 977.53,A -85,B 0,C 180,E1 24232.564,E2 24232.564} C_VEL
LIN {X 0,Y 245.823,Z 977.634,A -85,B 0,C 180,E1 24241.131,E2 24241.131} C_VEL
LIN {X 0,Y 268.106,Z 1032.205,A -85,B 0,C 180,E1 24247.777,E2 24247.777} C_VEL
LIN {X 0,Y 281.3,Z 1072.548,A -85,B 0,C 180,E1 24252.574,E2 24252.574} C_VEL
LIN {X 0,Y 288.096,Z 1099.167,A -85,B 0,C 180,E1 24255.944,E2 24255.944} C_VEL
LIN {X 0,Y 278.434,Z 1138.521,A -85,B 0,C 180,E1 24260.226,E2 24260.226} C_VEL
LIN {X 0,Y 268.71,Z 1173.774,A -85,B 0,C 180,E1 24265.651,E2 24265.651} C_VEL
LIN {X 0,Y 260.16,Z 1204.272,A -85,B 0,C 180,E1 24272.205,E2 24272.205} C_VEL
LIN {X 0,Y 254.111,Z 1228.494,A -85,B 0,C 180,E1 24279.469,E2 24279.469} C_VEL
LIN {X 0,Y 250.668,Z 1246.352,A -85,B 0,C 180,E1 24286.874,E2 24286.874} C_VEL
LIN {X 0,Y 249.206,Z 1259.566,A -85,B 0,C 180,E1 24294.743,E2 24294.743} C_VEL
LIN {X 0,Y 249.216,Z 1267.094,A -85,B 0,C 180,E1 24301.717,E2 24301.717} C_VEL
LIN {X 0,Y 251.09,Z 1271.961,A -85,B 0,C 180,E1 24310.404,E2 24310.404} C_VEL
LIN {X 0,Y 258.291,Z 1271.927,A -85,B 0,C 180,E1 24320.581,E2 24320.581} C_VEL
LIN {X 0,Y 272.569,Z 1266.264,A -85,B 0,C 180,E1 24329.991,E2 24329.991} C_VEL
LIN {X 0,Y 296.122,Z 1254.536,A -85,B 0,C 180,E1 24338.785,E2 24338.785} C_VEL
LIN {X 0,Y 312.092,Z 1245.96,A -85,B 0,C 180,E1 24342.789,E2 24342.789} C_VEL
LIN {X 0,Y 313.773,Z 1245.205,A -85,B 0,C 180,E1 24343.602,E2 24343.602} C_VEL
LIN {X 0,Y 284.305,Z 1265.045,A -85,B 0,C 180,E1 24351.245,E2 24351.245} C_VEL
LIN {X 0,Y 263.554,Z 1279.848,A -85,B 0,C 180,E1 24360.763,E2 24360.763} C_VEL
LIN {X 0,Y 254.016,Z 1287.177,A -85,B 0,C 180,E1 24369.045,E2 24369.045} C_VEL
LIN {X 0,Y 249.452,Z 1290.629,A -85,B 0,C 180,E1 24379.517,E2 24379.517} C_VEL
LIN {X 0,Y 249.366,Z 1289.172,A -85,B 0,C 180,E1 24386.533,E2 24386.533} C_VEL
LIN {X 0,Y 249.773,Z 1285.507,A -85,B 0,C 180,E1 24391.928,E2 24391.928} C_VEL
LIN {X 0,Y 249.958,Z 1277.338,A -85,B 0,C 180,E1 24398.733,E2 24398.733} C_VEL
LIN {X 0,Y 251.038,Z 1265.272,A -85,B 0,C 180,E1 24405.595,E2 24405.595} C_VEL
LIN {X 0,Y 256.367,Z 1255.969,A -85,B 0,C 180,E1 24415.391,E2 24415.391} C_VEL
LIN {X 0,Y 269.77,Z 1239.621,A -85,B 0,C 180,E1 24424.903,E2 24424.903} C_VEL
LIN {X 0,Y 289.972,Z 1217.231,A -85,B 0,C 180,E1 24432.81,E2 24432.81} C_VEL
LIN {X 0,Y 311.643,Z 1192.52,A -85,B 0,C 180,E1 24438.399,E2 24438.399} C_VEL
LIN {X 0,Y 335.475,Z 1162.706,A -85,B 0,C 180,E1 24442.777,E2 24442.777} C_VEL
LIN {X 0,Y 351.521,Z 1139.929,A -85,B 0,C 180,E1 24445.006,E2 24445.006} C_VEL
LIN {X 0,Y 351.703,Z 1139.135,A -85,B 0,C 180,E1 24445.964,E2 24445.964} C_VEL
LIN {X 0,Y 351.077,Z 1139.842,A -85,B 0,C 180,E1 24447.375,E2 24447.375} C_VEL
LIN {X 0,Y 330.776,Z 1166.266,A -85,B 0,C 180,E1 24450.527,E2 24450.527} C_VEL
LIN {X 0,Y 309.955,Z 1188.516,A -85,B 0,C 180,E1 24454.855,E2 24454.855} C_VEL
LIN {X 0,Y 290.543,Z 1205.258,A -85,B 0,C 180,E1 24460.291,E2 24460.291} C_VEL
LIN {X 0,Y 276.626,Z 1214.562,A -85,B 0,C 180,E1 24465.755,E2 24465.755} C_VEL
LIN {X 0,Y 268.087,Z 1218.565,A -85,B 0,C 180,E1 24470.262,E2 24470.262} C_VEL
LIN {X 0,Y 259.435,Z 1219.964,A -85,B 0,C 180,E1 24476.676,E2 24476.676} C_VEL
LIN {X 0,Y 253.952,Z 1216.692,A -85,B 0,C 180,E1 24483.445,E2 24483.445} C_VEL
LIN {X 0,Y 251.664,Z 1208.384,A -85,B 0,C 180,E1 24490.43,E2 24490.43} C_VEL
LIN {X 0,Y 251.6,Z 1203.635,A -85,B 0,C 180,E1 24493.142,E2 24493.142} C_VEL
LIN {X 0,Y 249.316,Z 1198.183,A -85,B 0,C 180,E1 24495.816,E2 24495.816} C_VEL
LIN {X 0,Y 244.957,Z 1188.524,A -85,B 0,C 180,E1 24499.723,E2 24499.723} C_VEL
LIN {X 0,Y 245.019,Z 1187.292,A -85,B 0,C 180,E1 24500.156,E2 24500.156} C_VEL
LIN {X 0,Y 247.944,Z 1166.422,A -85,B 0,C 180,E1 24506.204,E2 24506.204} C_VEL
LIN {X 0,Y 252.34,Z 1139.998,A -85,B 0,C 180,E1 24511.469,E2 24511.469} C_VEL
LIN {X 0,Y 256.95,Z 1109.709,A -85,B 0,C 180,E1 24515.536,E2 24515.536} C_VEL
LIN {X 0,Y 260.707,Z 1076.234,A -85,B 0,C 180,E1 24518.364,E2 24518.364} C_VEL
LIN {X 0,Y 261.502,Z 1059.458,A -85,B 0,C 180,E1 24519.526,E2 24519.526} C_VEL
LIN {X 0,Y 247.254,Z 1007.163,A -85,B 0,C 180,E1 24524.544,E2 24524.544} C_VEL
LIN {X 0,Y 237.427,Z 977.53,A -85,B 0,C 180,E1 24527.938,E2 24527.938} C_VEL
LIN {X 0,Y 237.5,Z 977.53,A -85,B 0,C 180,E1 24536.074,E2 24536.074} C_VEL
LIN {X 0,Y 237.939,Z 977.53,A -85,B 0,C 180,E1 24543.508,E2 24543.508} C_VEL
LIN {X 0,Y 238.792,Z 977.53,A -85,B 0,C 180,E1 24552.208,E2 24552.208} C_VEL
LIN {X 0,Y 239.426,Z 977.53,A -85,B 0,C 180,E1 24559.038,E2 24559.038} C_VEL
LIN {X 0,Y 240.307,Z 977.53,A -85,B 0,C 180,E1 24566.368,E2 24566.368} C_VEL
LIN {X 0,Y 240.745,Z 977.53,A -85,B 0,C 180,E1 24569.983,E2 24569.983} C_VEL
LIN {X 0,Y 239.794,Z 977.53,A -85,B 0,C 180,E1 24577.244,E2 24577.244} C_VEL
LIN {X 0,Y 238.981,Z 977.53,A -85,B 0,C 180,E1 24584.674,E2 24584.674} C_VEL
LIN {X 0,Y 238.352,Z 977.53,A -85,B 0,C 180,E1 24592.404,E2 24592.404} C_VEL
LIN {X 0,Y 237.888,Z 977.53,A -85,B 0,C 180,E1 24599.755,E2 24599.755} C_VEL
LIN {X 0,Y 259.741,Z 1030.687,A -85,B 0,C 180,E1 24606.574,E2 24606.574} C_VEL
LIN {X 0,Y 272.511,Z 1069.086,A -85,B 0,C 180,E1 24611.302,E2 24611.302} C_VEL
LIN {X 0,Y 280.651,Z 1100.476,A -85,B 0,C 180,E1 24615.397,E2 24615.397} C_VEL
LIN {X 0,Y 270.559,Z 1140.323,A -85,B 0,C 180,E1 24619.881,E2 24619.881} C_VEL
LIN {X 0,Y 260.681,Z 1175.219,A -85,B 0,C 180,E1 24625.453,E2 24625.453} C_VEL
LIN {X 0,Y 252.077,Z 1205.404,A -85,B 0,C 180,E1 24632.21,E2 24632.21} C_VEL
LIN {X 0,Y 246.025,Z 1229.45,A -85,B 0,C 180,E1 24639.706,E2 24639.706} C_VEL
LIN {X 0,Y 242.639,Z 1247.142,A -85,B 0,C 180,E1 24647.35,E2 24647.35} C_VEL
LIN {X 0,Y 241.26,Z 1260.212,A -85,B 0,C 180,E1 24655.472,E2 24655.472} C_VEL
LIN {X 0,Y 241.499,Z 1268.396,A -85,B 0,C 180,E1 24663.571,E2 24663.571} C_VEL
LIN {X 0,Y 243.303,Z 1272.297,A -85,B 0,C 180,E1 24670.741,E2 24670.741} C_VEL
LIN {X 0,Y 250.928,Z 1272.845,A -85,B 0,C 180,E1 24681.214,E2 24681.214} C_VEL
LIN {X 0,Y 265.883,Z 1267.904,A -85,B 0,C 180,E1 24690.827,E2 24690.827} C_VEL
LIN {X 0,Y 292.591,Z 1256.079,A -85,B 0,C 180,E1 24700.308,E2 24700.308} C_VEL
LIN {X 0,Y 304.718,Z 1250.279,A -85,B 0,C 180,E1 24703.24,E2 24703.24} C_VEL
LIN {X 0,Y 272.574,Z 1270.165,A -85,B 0,C 180,E1 24712.321,E2 24712.321} C_VEL
LIN {X 0,Y 254.216,Z 1282.063,A -85,B 0,C 180,E1 24721.539,E2 24721.539} C_VEL
LIN {X 0,Y 244.102,Z 1288.843,A -85,B 0,C 180,E1 24731.936,E2 24731.936} C_VEL
LIN {X 0,Y 241.627,Z 1290.073,A -85,B 0,C 180,E1 24739.173,E2 24739.173} C_VEL
LIN {X 0,Y 241.707,Z 1287.258,A -85,B 0,C 180,E1 24748.22,E2 24748.22} C_VEL
LIN {X 0,Y 242.077,Z 1280.776,A -85,B 0,C 180,E1 24755.404,E2 24755.404} C_VEL
LIN {X 0,Y 242.736,Z 1268.077,A -85,B 0,C 180,E1 24763.555,E2 24763.555} C_VEL
LIN {X 0,Y 243.161,Z 1264.686,A -85,B 0,C 180,E1 24765.568,E2 24765.568} C_VEL
LIN {X 0,Y 249.073,Z 1255.589,A -85,B 0,C 180,E1 24776.19,E2 24776.19} C_VEL
LIN {X 0,Y 262.125,Z 1241.14,A -85,B 0,C 180,E1 24785.334,E2 24785.334} C_VEL
LIN {X 0,Y 283.207,Z 1219.654,A -85,B 0,C 180,E1 24793.56,E2 24793.56} C_VEL
LIN {X 0,Y 306.697,Z 1194.948,A -85,B 0,C 180,E1 24799.45,E2 24799.45} C_VEL
LIN {X 0,Y 331.134,Z 1166.564,A -85,B 0,C 180,E1 24803.777,E2 24803.777} C_VEL
LIN {X 0,Y 346.703,Z 1146.12,A -85,B 0,C 180,E1 24805.872,E2 24805.872} C_VEL
LIN {X 0,Y 346.186,Z 1146.582,A -85,B 0,C 180,E1 24806.587,E2 24806.587} C_VEL
LIN {X 0,Y 324.483,Z 1172.366,A -85,B 0,C 180,E1 24809.897,E2 24809.897} C_VEL
LIN {X 0,Y 302.37,Z 1193.792,A -85,B 0,C 180,E1 24814.457,E2 24814.457} C_VEL
LIN {X 0,Y 283.382,Z 1208.497,A -85,B 0,C 180,E1 24819.771,E2 24819.771} C_VEL
LIN {X 0,Y 269.131,Z 1216.924,A -85,B 0,C 180,E1 24825.349,E2 24825.349} C_VEL
LIN {X 0,Y 260.384,Z 1220.361,A -85,B 0,C 180,E1 24829.971,E2 24829.971} C_VEL
LIN {X 0,Y 251.521,Z 1221.034,A -85,B 0,C 180,E1 24836.571,E2 24836.571} C_VEL
LIN {X 0,Y 245.958,Z 1217.045,A -85,B 0,C 180,E1 24843.557,E2 24843.557} C_VEL
LIN {X 0,Y 243.758,Z 1208.001,A -85,B 0,C 180,E1 24850.772,E2 24850.772} C_VEL
LIN {X 0,Y 244.425,Z 1192.913,A -85,B 0,C 180,E1 24858.082,E2 24858.082} C_VEL
LIN {X 0,Y 245.019,Z 1187.292,A -85,B 0,C 180,E1 24860.156,E2 24860.156} C_VEL
LIN {X 0,Y 243.478,Z 1179.766,A -85,B 0,C 180,E1 24862.658,E2 24862.658} C_VEL
LIN {X 0,Y 240.054,Z 1167.278,A -85,B 0,C 180,E1 24866.229,E2 24866.229} C_VEL
LIN {X 0,Y 240.224,Z 1165.741,A -85,B 0,C 180,E1 24866.608,E2 24866.608} C_VEL
LIN {X 0,Y 244.591,Z 1140.242,A -85,B 0,C 180,E1 24871.801,E2 24871.801} C_VEL
LIN {X 0,Y 249.292,Z 1109.954,A -85,B 0,C 180,E1 24875.965,E2 24875.965} C_VEL
LIN {X 0,Y 253.344,Z 1074.689,A -85,B 0,C 180,E1 24879.008,E2 24879.008} C_VEL
LIN {X 0,Y 253.964,Z 1060.814,A -85,B 0,C 180,E1 24880.024,E2 24880.024} C_VEL
LIN {X 0,Y 240.207,Z 1009.902,A -85,B 0,C 180,E1 24885.088,E2 24885.088} C_VEL
LIN {X 0,Y 229.431,Z 977.53,A -85,B 0,C 180,E1 24888.903,E2 24888.903} C_VEL
LIN {X 0,Y 229.725,Z 977.53,A -85,B 0,C 180,E1 24899.076,E2 24899.076} C_VEL
LIN {X 0,Y 230.386,Z 977.53,A -85,B 0,C 180,E1 24907.095,E2 24907.095} C_VEL
LIN {X 0,Y 231.013,Z 977.53,A -85,B 0,C 180,E1 24914.771,E2 24914.771} C_VEL
LIN {X 0,Y 231.847,Z 977.53,A -85,B 0,C 180,E1 24922.472,E2 24922.472} C_VEL
LIN {X 0,Y 232.832,Z 977.53,A -85,B 0,C 180,E1 24929.983,E2 24929.983} C_VEL
LIN {X 0,Y 231.825,Z 977.53,A -85,B 0,C 180,E1 24937.494,E2 24937.494} C_VEL
LIN {X 0,Y 230.997,Z 977.53,A -85,B 0,C 180,E1 24945.194,E2 24945.194} C_VEL
LIN {X 0,Y 230.273,Z 977.53,A -85,B 0,C 180,E1 24953.236,E2 24953.236} C_VEL
LIN {X 0,Y 229.987,Z 977.901,A -85,B 0,C 180,E1 24958.36,E2 24958.36} C_VEL
LIN {X 0,Y 251.648,Z 1029.81,A -85,B 0,C 180,E1 24965.4,E2 24965.4} C_VEL
LIN {X 0,Y 264.768,Z 1069.333,A -85,B 0,C 180,E1 24970.449,E2 24970.449} C_VEL
LIN {X 0,Y 273.184,Z 1101.914,A -85,B 0,C 180,E1 24974.846,E2 24974.846} C_VEL
LIN {X 0,Y 262.803,Z 1141.492,A -85,B 0,C 180,E1 24979.447,E2 24979.447} C_VEL
LIN {X 0,Y 252.669,Z 1176.596,A -85,B 0,C 180,E1 24985.244,E2 24985.244} C_VEL
LIN {X 0,Y 243.967,Z 1206.468,A -85,B 0,C 180,E1 24992.211,E2 24992.211} C_VEL
LIN {X 0,Y 237.873,Z 1230.337,A -85,B 0,C 180,E1 24999.952,E2 24999.952} C_VEL
LIN {X 0,Y 234.615,Z 1247.882,A -85,B 0,C 180,E1 25007.858,E2 25007.858} C_VEL
LIN {X 0,Y 233.327,Z 1260.826,A -85,B 0,C 180,E1 25016.25,E2 25016.25} C_VEL
LIN {X 0,Y 233.609,Z 1268.226,A -85,B 0,C 180,E1 25023.692,E2 25023.692} C_VEL
LIN {X 0,Y 237.428,Z 1273.547,A -85,B 0,C 180,E1 25034.761,E2 25034.761} C_VEL
LIN {X 0,Y 247.982,Z 1272.893,A -85,B 0,C 180,E1 25045.293,E2 25045.293} C_VEL
LIN {X 0,Y 266.196,Z 1267.074,A -85,B 0,C 180,E1 25054.663,E2 25054.663} C_VEL
LIN {X 0,Y 294.712,Z 1255.482,A -85,B 0,C 180,E1 25063.355,E2 25063.355} C_VEL
LIN {X 0,Y 266.407,Z 1271.35,A -85,B 0,C 180,E1 25071.289,E2 25071.289} C_VEL
LIN {X 0,Y 247.189,Z 1282.379,A -85,B 0,C 180,E1 25080.652,E2 25080.652} C_VEL
LIN {X 0,Y 236.489,Z 1288.509,A -85,B 0,C 180,E1 25091.333,E2 25091.333} C_VEL
LIN {X 0,Y 233.499,Z 1288.727,A -85,B 0,C 180,E1 25102.56,E2 25102.56} C_VEL
LIN {X 0,Y 234.223,Z 1284.925,A -85,B 0,C 180,E1 25110.017,E2 25110.017} C_VEL
LIN {X 0,Y 234.287,Z 1277.034,A -85,B 0,C 180,E1 25117.449,E2 25117.449} C_VEL
LIN {X 0,Y 235.234,Z 1264.223,A -85,B 0,C 180,E1 25125.06,E2 25125.06} C_VEL
LIN {X 0,Y 239.729,Z 1257.584,A -85,B 0,C 180,E1 25134.777,E2 25134.777} C_VEL
LIN {X 0,Y 252.61,Z 1244.379,A -85,B 0,C 180,E1 25144.759,E2 25144.759} C_VEL
LIN {X 0,Y 272.272,Z 1225.925,A -85,B 0,C 180,E1 25153,E2 25153} C_VEL
LIN {X 0,Y 297.891,Z 1201.243,A -85,B 0,C 180,E1 25159.75,E2 25159.75} C_VEL
LIN {X 0,Y 323.996,Z 1173.661,A -85,B 0,C 180,E1 25164.371,E2 25164.371} C_VEL
LIN {X 0,Y 336.015,Z 1159.535,A -85,B 0,C 180,E1 25166.018,E2 25166.018} C_VEL
LIN {X 0,Y 337.081,Z 1158.124,A -85,B 0,C 180,E1 25166.352,E2 25166.352} C_VEL
LIN {X 0,Y 314.788,Z 1181.544,A -85,B 0,C 180,E1 25169.855,E2 25169.855} C_VEL
LIN {X 0,Y 292.688,Z 1200.406,A -85,B 0,C 180,E1 25174.558,E2 25174.558} C_VEL
LIN {X 0,Y 272.439,Z 1213.848,A -85,B 0,C 180,E1 25180.532,E2 25180.532} C_VEL
LIN {X 0,Y 258.436,Z 1220.387,A -85,B 0,C 180,E1 25186.463,E2 25186.463} C_VEL
LIN {X 0,Y 247.723,Z 1222.531,A -85,B 0,C 180,E1 25192.999,E2 25192.999} C_VEL
LIN {X 0,Y 240.37,Z 1220.221,A -85,B 0,C 180,E1 25200.026,E2 25200.026} C_VEL
LIN {X 0,Y 236.252,Z 1211.834,A -85,B 0,C 180,E1 25208.323,E2 25208.323} C_VEL
LIN {X 0,Y 236.128,Z 1197.932,A -85,B 0,C 180,E1 25216.09,E2 25216.09} C_VEL
LIN {X 0,Y 238.337,Z 1178.471,A -85,B 0,C 180,E1 25223.167,E2 25223.167} C_VEL
LIN {X 0,Y 240.224,Z 1165.741,A -85,B 0,C 180,E1 25226.608,E2 25226.608} C_VEL
LIN {X 0,Y 237.683,Z 1157.729,A -85,B 0,C 180,E1 25228.598,E2 25228.598} C_VEL
LIN {X 0,Y 235.331,Z 1149.181,A -85,B 0,C 180,E1 25230.52,E2 25230.52} C_VEL
LIN {X 0,Y 240.008,Z 1120.232,A -85,B 0,C 180,E1 25235.203,E2 25235.203} C_VEL
LIN {X 0,Y 244.501,Z 1087.731,A -85,B 0,C 180,E1 25238.574,E2 25238.574} C_VEL
LIN {X 0,Y 246.431,Z 1062.251,A -85,B 0,C 180,E1 25240.506,E2 25240.506} C_VEL
LIN {X 0,Y 233.011,Z 1012.177,A -85,B 0,C 180,E1 25245.718,E2 25245.718} C_VEL
LIN {X 0,Y 221.492,Z 977.53,A -85,B 0,C 180,E1 25249.963,E2 25249.963} C_VEL
LIN {X 0,Y 221.46,Z 977.53,A -85,B 0,C 180,E1 25256.791,E2 25256.791} C_VEL
LIN {X 0,Y 222.198,Z 977.53,A -85,B 0,C 180,E1 25265.828,E2 25265.828} C_VEL
LIN {X 0,Y 222.986,Z 977.53,A -85,B 0,C 180,E1 25274.209,E2 25274.209} C_VEL
LIN {X 0,Y 223.898,Z 977.53,A -85,B 0,C 180,E1 25282.203,E2 25282.203} C_VEL
LIN {X 0,Y 224.926,Z 977.53,A -85,B 0,C 180,E1 25289.982,E2 25289.982} C_VEL
LIN {X 0,Y 223.876,Z 977.53,A -85,B 0,C 180,E1 25297.762,E2 25297.762} C_VEL
LIN {X 0,Y 222.749,Z 977.53,A -85,B 0,C 180,E1 25307.687,E2 25307.687} C_VEL
LIN {X 0,Y 222.067,Z 977.558,A -85,B 0,C 180,E1 25316.805,E2 25316.805} C_VEL
LIN {X 0,Y 244.103,Z 1030.197,A -85,B 0,C 180,E1 25324.347,E2 25324.347} C_VEL
LIN {X 0,Y 257.073,Z 1069.687,A -85,B 0,C 180,E1 25329.572,E2 25329.572} C_VEL
LIN {X 0,Y 265.636,Z 1103.576,A -85,B 0,C 180,E1 25334.309,E2 25334.309} C_VEL
LIN {X 0,Y 255.172,Z 1142.387,A -85,B 0,C 180,E1 25338.963,E2 25338.963} C_VEL
LIN {X 0,Y 244.7,Z 1177.836,A -85,B 0,C 180,E1 25345.029,E2 25345.029} C_VEL
LIN {X 0,Y 235.831,Z 1207.463,A -85,B 0,C 180,E1 25352.21,E2 25352.21} C_VEL
LIN {X 0,Y 229.749,Z 1231.163,A -85,B 0,C 180,E1 25360.218,E2 25360.218} C_VEL
LIN {X 0,Y 226.578,Z 1248.569,A -85,B 0,C 180,E1 25368.4,E2 25368.4} C_VEL
LIN {X 0,Y 225.412,Z 1261.401,A -85,B 0,C 180,E1 25377.083,E2 25377.083} C_VEL
LIN {X 0,Y 225.984,Z 1269.473,A -85,B 0,C 180,E1 25385.744,E2 25385.744} C_VEL
LIN {X 0,Y 229.785,Z 1273.879,A -85,B 0,C 180,E1 25395.264,E2 25395.264} C_VEL
LIN {X 0,Y 240.884,Z 1273.865,A -85,B 0,C 180,E1 25406.093,E2 25406.093} C_VEL
LIN {X 0,Y 263.864,Z 1267.6,A -85,B 0,C 180,E1 25417.049,E2 25417.049} C_VEL
LIN {X 0,Y 283.374,Z 1260.603,A -85,B 0,C 180,E1 25422.75,E2 25422.75} C_VEL
LIN {X 0,Y 284.07,Z 1260.459,A -85,B 0,C 180,E1 25423.432,E2 25423.432} C_VEL
LIN {X 0,Y 256.429,Z 1274.489,A -85,B 0,C 180,E1 25431.671,E2 25431.671} C_VEL
LIN {X 0,Y 237.774,Z 1283.983,A -85,B 0,C 180,E1 25441.468,E2 25441.468} C_VEL
LIN {X 0,Y 228.886,Z 1288.171,A -85,B 0,C 180,E1 25450.689,E2 25450.689} C_VEL
LIN {X 0,Y 225.647,Z 1287.88,A -85,B 0,C 180,E1 25462.3,E2 25462.3} C_VEL
LIN {X 0,Y 226.393,Z 1283.803,A -85,B 0,C 180,E1 25470.018,E2 25470.018} C_VEL
LIN {X 0,Y 226.462,Z 1275.446,A -85,B 0,C 180,E1 25477.708,E2 25477.708} C_VEL
LIN {X 0,Y 227.427,Z 1263.251,A -85,B 0,C 180,E1 25485.475,E2 25485.475} C_VEL
LIN {X 0,Y 231.997,Z 1257.436,A -85,B 0,C 180,E1 25495.141,E2 25495.141} C_VEL
LIN {X 0,Y 244.54,Z 1245.847,A -85,B 0,C 180,E1 25504.991,E2 25504.991} C_VEL
LIN {X 0,Y 264.485,Z 1228.755,A -85,B 0,C 180,E1 25513.453,E2 25513.453} C_VEL
LIN {X 0,Y 290.391,Z 1205.89,A -85,B 0,C 180,E1 25520.345,E2 25520.345} C_VEL
LIN {X 0,Y 319.798,Z 1177.248,A -85,B 0,C 180,E1 25525.432,E2 25525.432} C_VEL
LIN {X 0,Y 325.635,Z 1170.927,A -85,B 0,C 180,E1 25526.415,E2 25526.415} C_VEL
LIN {X 0,Y 302.193,Z 1192.142,A -85,B 0,C 180,E1 25530.348,E2 25530.348} C_VEL
LIN {X 0,Y 280.541,Z 1207.921,A -85,B 0,C 180,E1 25535.282,E2 25535.282} C_VEL
LIN {X 0,Y 261.34,Z 1218.481,A -85,B 0,C 180,E1 25541.431,E2 25541.431} C_VEL
LIN {X 0,Y 248.723,Z 1222.893,A -85,B 0,C 180,E1 25547.169,E2 25547.169} C_VEL
LIN {X 0,Y 239.869,Z 1223.736,A -85,B 0,C 180,E1 25552.769,E2 25552.769} C_VEL
LIN {X 0,Y 232.387,Z 1220.686,A -85,B 0,C 180,E1 25560.027,E2 25560.027} C_VEL
LIN {X 0,Y 228.286,Z 1211.525,A -85,B 0,C 180,E1 25568.615,E2 25568.615} C_VEL
LIN {X 0,Y 228.231,Z 1197.918,A -85,B 0,C 180,E1 25576.139,E2 25576.139} C_VEL
LIN {X 0,Y 230.456,Z 1178.757,A -85,B 0,C 180,E1 25583.261,E2 25583.261} C_VEL
LIN {X 0,Y 234.294,Z 1154.653,A -85,B 0,C 180,E1 25589.408,E2 25589.408} C_VEL
LIN {X 0,Y 235.331,Z 1149.181,A -85,B 0,C 180,E1 25590.52,E2 25590.52} C_VEL
LIN {X 0,Y 234.67,Z 1138.929,A -85,B 0,C 180,E1 25592.521,E2 25592.521} C_VEL
LIN {X 0,Y 232.006,Z 1122.826,A -85,B 0,C 180,E1 25595.297,E2 25595.297} C_VEL
LIN {X 0,Y 232.227,Z 1120.896,A -85,B 0,C 180,E1 25595.566,E2 25595.566} C_VEL
LIN {X 0,Y 236.737,Z 1090.037,A -85,B 0,C 180,E1 25598.935,E2 25598.935} C_VEL
LIN {X 0,Y 239.262,Z 1065.248,A -85,B 0,C 180,E1 25600.86,E2 25600.86} C_VEL
LIN {X 0,Y 226.066,Z 1015.109,A -85,B 0,C 180,E1 25606.288,E2 25606.288} C_VEL
LIN {X 0,Y 213.515,Z 977.53,A -85,B 0,C 180,E1 25611.072,E2 25611.072} C_VEL
LIN {X 0,Y 213.722,Z 977.53,A -85,B 0,C 180,E1 25620.223,E2 25620.223} C_VEL
LIN {X 0,Y 214.552,Z 977.53,A -85,B 0,C 180,E1 25629.302,E2 25629.302} C_VEL
LIN {X 0,Y 215.422,Z 977.53,A -85,B 0,C 180,E1 25637.799,E2 25637.799} C_VEL
LIN {X 0,Y 216.457,Z 977.53,A -85,B 0,C 180,E1 25645.967,E2 25645.967} C_VEL
LIN {X 0,Y 217.009,Z 977.53,A -85,B 0,C 180,E1 25649.981,E2 25649.981} C_VEL
LIN {X 0,Y 215.893,Z 977.53,A -85,B 0,C 180,E1 25658.05,E2 25658.05} C_VEL
LIN {X 0,Y 214.968,Z 977.53,A -85,B 0,C 180,E1 25666.357,E2 25666.357} C_VEL
LIN {X 0,Y 214.208,Z 977.533,A -85,B 0,C 180,E1 25675.195,E2 25675.195} C_VEL
LIN {X 0,Y 235.936,Z 1029.226,A -85,B 0,C 180,E1 25683.031,E2 25683.031} C_VEL
LIN {X 0,Y 248.711,Z 1067.806,A -85,B 0,C 180,E1 25688.344,E2 25688.344} C_VEL
LIN {X 0,Y 258.051,Z 1103.534,A -85,B 0,C 180,E1 25693.532,E2 25693.532} C_VEL
LIN {X 0,Y 247.854,Z 1142.147,A -85,B 0,C 180,E1 25698.302,E2 25698.302} C_VEL
LIN {X 0,Y 237.04,Z 1177.922,A -85,B 0,C 180,E1 25704.57,E2 25704.57} C_VEL
LIN {X 0,Y 228.194,Z 1206.796,A -85,B 0,C 180,E1 25711.736,E2 25711.736} C_VEL
LIN {X 0,Y 221.915,Z 1230.738,A -85,B 0,C 180,E1 25720.01,E2 25720.01} C_VEL
LIN {X 0,Y 218.542,Z 1249.21,A -85,B 0,C 180,E1 25728.98,E2 25728.98} C_VEL
LIN {X 0,Y 217.558,Z 1261.94,A -85,B 0,C 180,E1 25737.976,E2 25737.976} C_VEL
LIN {X 0,Y 218.536,Z 1270.645,A -85,B 0,C 180,E1 25747.942,E2 25747.942} C_VEL
LIN {X 0,Y 225.091,Z 1275.017,A -85,B 0,C 180,E1 25759.638,E2 25759.638} C_VEL
LIN {X 0,Y 239.584,Z 1273.939,A -85,B 0,C 180,E1 25770.361,E2 25770.361} C_VEL
LIN {X 0,Y 266.487,Z 1266.839,A -85,B 0,C 180,E1 25780.8,E2 25780.8} C_VEL
LIN {X 0,Y 274.237,Z 1264.375,A -85,B 0,C 180,E1 25782.902,E2 25782.902} C_VEL
LIN {X 0,Y 272.59,Z 1265.272,A -85,B 0,C 180,E1 25783.749,E2 25783.749} C_VEL
LIN {X 0,Y 242.731,Z 1278.823,A -85,B 0,C 180,E1 25793.648,E2 25793.648} C_VEL
LIN {X 0,Y 224.31,Z 1286.805,A -85,B 0,C 180,E1 25806.109,E2 25806.109} C_VEL
LIN {X 0,Y 218.199,Z 1287.993,A -85,B 0,C 180,E1 25817.994,E2 25817.994} C_VEL
LIN {X 0,Y 218.228,Z 1283.958,A -85,B 0,C 180,E1 25828.029,E2 25828.029} C_VEL
LIN {X 0,Y 218.637,Z 1277.636,A -85,B 0,C 180,E1 25834.988,E2 25834.988} C_VEL
LIN {X 0,Y 219.288,Z 1265.045,A -85,B 0,C 180,E1 25843.53,E2 25843.53} C_VEL
LIN {X 0,Y 219.554,Z 1262.446,A -85,B 0,C 180,E1 25845.069,E2 25845.069} C_VEL
LIN {X 0,Y 224.69,Z 1256.856,A -85,B 0,C 180,E1 25856.018,E2 25856.018} C_VEL
LIN {X 0,Y 239.555,Z 1244.638,A -85,B 0,C 180,E1 25866.956,E2 25866.956} C_VEL
LIN {X 0,Y 262.842,Z 1226.463,A -85,B 0,C 180,E1 25875.918,E2 25875.918} C_VEL
LIN {X 0,Y 289.681,Z 1204.436,A -85,B 0,C 180,E1 25882.317,E2 25882.317} C_VEL
LIN {X 0,Y 312.815,Z 1183.452,A -85,B 0,C 180,E1 25886.122,E2 25886.122} C_VEL
LIN {X 0,Y 313.411,Z 1182.766,A -85,B 0,C 180,E1 25886.601,E2 25886.601} C_VEL
LIN {X 0,Y 288.921,Z 1201.773,A -85,B 0,C 180,E1 25891.008,E2 25891.008} C_VEL
LIN {X 0,Y 266.632,Z 1215.222,A -85,B 0,C 180,E1 25896.587,E2 25896.587} C_VEL
LIN {X 0,Y 250.184,Z 1222.266,A -85,B 0,C 180,E1 25902.401,E2 25902.401} C_VEL
LIN {X 0,Y 237.182,Z 1225.033,A -85,B 0,C 180,E1 25908.978,E2 25908.978} C_VEL
LIN {X 0,Y 227.705,Z 1223.52,A -85,B 0,C 180,E1 25916.212,E2 25916.212} C_VEL
LIN {X 0,Y 221.456,Z 1216.003,A -85,B 0,C 180,E1 25925.194,E2 25925.194} C_VEL
LIN {X 0,Y 220.107,Z 1202.919,A -85,B 0,C 180,E1 25933.736,E2 25933.736} C_VEL
LIN {X 0,Y 221.706,Z 1185.115,A -85,B 0,C 180,E1 25941.312,E2 25941.312} C_VEL
LIN {X 0,Y 225.347,Z 1161.714,A -85,B 0,C 180,E1 25948.107,E2 25948.107} C_VEL
LIN {X 0,Y 230.14,Z 1134.167,A -85,B 0,C 180,E1 25953.577,E2 25953.577} C_VEL
LIN {X 0,Y 232.227,Z 1120.896,A -85,B 0,C 180,E1 25955.566,E2 25955.566} C_VEL
LIN {X 0,Y 230.755,Z 1105.647,A -85,B 0,C 180,E1 25957.69,E2 25957.69} C_VEL
LIN {X 0,Y 229.198,Z 1089.765,A -85,B 0,C 180,E1 25959.517,E2 25959.517} C_VEL
LIN {X 0,Y 231.325,Z 1065.076,A -85,B 0,C 180,E1 25961.574,E2 25961.574} C_VEL
LIN {X 0,Y 219.014,Z 1017.867,A -85,B 0,C 180,E1 25966.88,E2 25966.88} C_VEL
LIN {X 0,Y 205.519,Z 977.53,A -85,B 0,C 180,E1 25972.317,E2 25972.317} C_VEL
LIN {X 0,Y 205.863,Z 977.53,A -85,B 0,C 180,E1 25982.09,E2 25982.09} C_VEL
LIN {X 0,Y 206.537,Z 977.53,A -85,B 0,C 180,E1 25988.459,E2 25988.459} C_VEL
LIN {X 0,Y 207.403,Z 977.53,A -85,B 0,C 180,E1 25997.319,E2 25997.319} C_VEL
LIN {X 0,Y 208.499,Z 977.53,A -85,B 0,C 180,E1 26005.813,E2 26005.813} C_VEL
LIN {X 0,Y 209.112,Z 977.53,A -85,B 0,C 180,E1 26009.981,E2 26009.981} C_VEL
LIN {X 0,Y 207.936,Z 977.53,A -85,B 0,C 180,E1 26018.361,E2 26018.361} C_VEL
LIN {X 0,Y 206.814,Z 977.53,A -85,B 0,C 180,E1 26027.659,E2 26027.659} C_VEL
LIN {X 0,Y 206.379,Z 977.936,A -85,B 0,C 180,E1 26033.511,E2 26033.511} C_VEL
LIN {X 0,Y 227.16,Z 1026.571,A -85,B 0,C 180,E1 26041.412,E2 26041.412} C_VEL
LIN {X 0,Y 240.328,Z 1065.493,A -85,B 0,C 180,E1 26047.011,E2 26047.011} C_VEL
LIN {X 0,Y 250.205,Z 1103.536,A -85,B 0,C 180,E1 26052.697,E2 26052.697} C_VEL
LIN {X 0,Y 249.659,Z 1110.066,A -85,B 0,C 180,E1 26053.529,E2 26053.529} C_VEL
LIN {X 0,Y 238.436,Z 1149.063,A -85,B 0,C 180,E1 26058.722,E2 26058.722} C_VEL
LIN {X 0,Y 227.719,Z 1183.062,A -85,B 0,C 180,E1 26065.238,E2 26065.238} C_VEL
LIN {X 0,Y 219.023,Z 1211.29,A -85,B 0,C 180,E1 26072.859,E2 26072.859} C_VEL
LIN {X 0,Y 213.256,Z 1233.827,A -85,B 0,C 180,E1 26081.324,E2 26081.324} C_VEL
LIN {X 0,Y 210.387,Z 1251.495,A -85,B 0,C 180,E1 26090.645,E2 26090.645} C_VEL
LIN {X 0,Y 209.784,Z 1263.523,A -85,B 0,C 180,E1 26099.97,E2 26099.97} C_VEL
LIN {X 0,Y 211.341,Z 1271.68,A -85,B 0,C 180,E1 26110.295,E2 26110.295} C_VEL
LIN {X 0,Y 217.629,Z 1275.48,A -85,B 0,C 180,E1 26120.34,E2 26120.34} C_VEL
LIN {X 0,Y 232.861,Z 1275.094,A -85,B 0,C 180,E1 26131.335,E2 26131.335} C_VEL
LIN {X 0,Y 260.79,Z 1268.995,A -85,B 0,C 180,E1 26141.889,E2 26141.889} C_VEL
LIN {X 0,Y 263.157,Z 1268.316,A -85,B 0,C 180,E1 26142.538,E2 26142.538} C_VEL
LIN {X 0,Y 263.979,Z 1268.239,A -85,B 0,C 180,E1 26143.346,E2 26143.346} C_VEL
LIN {X 0,Y 232.833,Z 1280.766,A -85,B 0,C 180,E1 26154.168,E2 26154.168} C_VEL
LIN {X 0,Y 217.013,Z 1286.494,A -85,B 0,C 180,E1 26165.253,E2 26165.253} C_VEL
LIN {X 0,Y 210.426,Z 1287.125,A -85,B 0,C 180,E1 26177.544,E2 26177.544} C_VEL
LIN {X 0,Y 210.414,Z 1282.78,A -85,B 0,C 180,E1 26187.956,E2 26187.956} C_VEL
LIN {X 0,Y 210.845,Z 1276.143,A -85,B 0,C 180,E1 26195.173,E2 26195.173} C_VEL
LIN {X 0,Y 211.666,Z 1262.184,A -85,B 0,C 180,E1 26204.516,E2 26204.516} C_VEL
LIN {X 0,Y 219.368,Z 1254.717,A -85,B 0,C 180,E1 26218.936,E2 26218.936} C_VEL
LIN {X 0,Y 237.128,Z 1241.999,A -85,B 0,C 180,E1 26229.981,E2 26229.981} C_VEL
LIN {X 0,Y 262.686,Z 1223.673,A -85,B 0,C 180,E1 26238.603,E2 26238.603} C_VEL
LIN {X 0,Y 289.386,Z 1203.139,A -85,B 0,C 180,E1 26244.276,E2 26244.276} C_VEL
LIN {X 0,Y 302.542,Z 1192.091,A -85,B 0,C 180,E1 26246.598,E2 26246.598} C_VEL
LIN {X 0,Y 277.11,Z 1209.134,A -85,B 0,C 180,E1 26251.418,E2 26251.418} C_VEL
LIN {X 0,Y 256.535,Z 1219.596,A -85,B 0,C 180,E1 26256.844,E2 26256.844} C_VEL
LIN {X 0,Y 242.783,Z 1224.375,A -85,B 0,C 180,E1 26261.846,E2 26261.846} C_VEL
LIN {X 0,Y 229.436,Z 1226.35,A -85,B 0,C 180,E1 26268.601,E2 26268.601} C_VEL
LIN {X 0,Y 219.742,Z 1224.099,A -85,B 0,C 180,E1 26276.075,E2 26276.075} C_VEL
LIN {X 0,Y 213.631,Z 1216.319,A -85,B 0,C 180,E1 26284.945,E2 26284.945} C_VEL
LIN {X 0,Y 212.196,Z 1203.762,A -85,B 0,C 180,E1 26293.25,E2 26293.25} C_VEL
LIN {X 0,Y 213.557,Z 1186.78,A -85,B 0,C 180,E1 26300.808,E2 26300.808} C_VEL
LIN {X 0,Y 216.892,Z 1164.807,A -85,B 0,C 180,E1 26307.599,E2 26307.599} C_VEL
LIN {X 0,Y 221.592,Z 1138.856,A -85,B 0,C 180,E1 26313.194,E2 26313.194} C_VEL
LIN {X 0,Y 226.841,Z 1107.383,A -85,B 0,C 180,E1 26317.736,E2 26317.736} C_VEL
LIN {X 0,Y 229.198,Z 1089.765,A -85,B 0,C 180,E1 26319.517,E2 26319.517} C_VEL
LIN {X 0,Y 228.126,Z 1077.578,A -85,B 0,C 180,E1 26320.74,E2 26320.74} C_VEL
LIN {X 0,Y 221.846,Z 1057.929,A -85,B 0,C 180,E1 26323.062,E2 26323.062} C_VEL
LIN {X 0,Y 209.349,Z 1011.814,A -85,B 0,C 180,E1 26328.639,E2 26328.639} C_VEL
LIN {X 0,Y 197.562,Z 977.53,A -85,B 0,C 180,E1 26333.656,E2 26333.656} C_VEL
LIN {X 0,Y 198.024,Z 977.53,A -85,B 0,C 180,E1 26342.647,E2 26342.647} C_VEL
LIN {X 0,Y 198.919,Z 977.53,A -85,B 0,C 180,E1 26352.239,E2 26352.239} C_VEL
LIN {X 0,Y 199.955,Z 977.53,A -85,B 0,C 180,E1 26361.262,E2 26361.262} C_VEL
LIN {X 0,Y 201.19,Z 977.53,A -85,B 0,C 180,E1 26369.98,E2 26369.98} C_VEL
LIN {X 0,Y 199.775,Z 977.53,A -85,B 0,C 180,E1 26379.441,E2 26379.441} C_VEL
LIN {X 0,Y 198.652,Z 977.53,A -85,B 0,C 180,E1 26390.053,E2 26390.053} C_VEL
LIN {X 0,Y 198.624,Z 977.794,A -85,B 0,C 180,E1 26391.664,E2 26391.664} C_VEL
LIN {X 0,Y 219.019,Z 1025.658,A -85,B 0,C 180,E1 26399.94,E2 26399.94} C_VEL
LIN {X 0,Y 231.644,Z 1062.27,A -85,B 0,C 180,E1 26405.467,E2 26405.467} C_VEL
LIN {X 0,Y 241.307,Z 1098.719,A -85,B 0,C 180,E1 26411.072,E2 26411.072} C_VEL
LIN {X 0,Y 242.694,Z 1109.2,A -85,B 0,C 180,E1 26412.667,E2 26412.667} C_VEL
LIN {X 0,Y 231.038,Z 1148.905,A -85,B 0,C 180,E1 26418.046,E2 26418.046} C_VEL
LIN {X 0,Y 220.049,Z 1182.951,A -85,B 0,C 180,E1 26424.751,E2 26424.751} C_VEL
LIN {X 0,Y 211.038,Z 1211.583,A -85,B 0,C 180,E1 26432.73,E2 26432.73} C_VEL
LIN {X 0,Y 205.145,Z 1234.474,A -85,B 0,C 180,E1 26441.675,E2 26441.675} C_VEL
LIN {X 0,Y 202.364,Z 1252.021,A -85,B 0,C 180,E1 26451.357,E2 26451.357} C_VEL
LIN {X 0,Y 201.933,Z 1263.971,A -85,B 0,C 180,E1 26461.044,E2 26461.044} C_VEL
LIN {X 0,Y 203.55,Z 1271.58,A -85,B 0,C 180,E1 26470.693,E2 26470.693} C_VEL
LIN {X 0,Y 210.203,Z 1275.794,A -85,B 0,C 180,E1 26481.092,E2 26481.092} C_VEL
LIN {X 0,Y 226.193,Z 1276.125,A -85,B 0,C 180,E1 26492.369,E2 26492.369} C_VEL
LIN {X 0,Y 254.025,Z 1271.239,A -85,B 0,C 180,E1 26502.725,E2 26502.725} C_VEL
LIN {X 0,Y 251.947,Z 1272.144,A -85,B 0,C 180,E1 26503.828,E2 26503.828} C_VEL
LIN {X 0,Y 223.885,Z 1281.971,A -85,B 0,C 180,E1 26514.251,E2 26514.251} C_VEL
LIN {X 0,Y 209.742,Z 1286.179,A -85,B 0,C 180,E1 26524.334,E2 26524.334} C_VEL
LIN {X 0,Y 202.676,Z 1286.22,A -85,B 0,C 180,E1 26537.059,E2 26537.059} C_VEL
LIN {X 0,Y 202.641,Z 1281.457,A -85,B 0,C 180,E1 26547.877,E2 26547.877} C_VEL
LIN {X 0,Y 203.074,Z 1274.476,A -85,B 0,C 180,E1 26555.372,E2 26555.372} C_VEL
LIN {X 0,Y 203.906,Z 1260.261,A -85,B 0,C 180,E1 26565.113,E2 26565.113} C_VEL
LIN {X 0,Y 210.238,Z 1255.52,A -85,B 0,C 180,E1 26577.957,E2 26577.957} C_VEL
LIN {X 0,Y 226.691,Z 1244.903,A -85,B 0,C 180,E1 26589.304,E2 26589.304} C_VEL
LIN {X 0,Y 252.843,Z 1228.059,A -85,B 0,C 180,E1 26598.678,E2 26598.678} C_VEL
LIN {X 0,Y 283.543,Z 1206.54,A -85,B 0,C 180,E1 26605.275,E2 26605.275} C_VEL
LIN {X 0,Y 290.968,Z 1200.917,A -85,B 0,C 180,E1 26606.457,E2 26606.457} C_VEL
LIN {X 0,Y 278.677,Z 1208.384,A -85,B 0,C 180,E1 26608.929,E2 26608.929} C_VEL
LIN {X 0,Y 257.44,Z 1219.14,A -85,B 0,C 180,E1 26613.834,E2 26613.834} C_VEL
LIN {X 0,Y 235.393,Z 1226.388,A -85,B 0,C 180,E1 26621.255,E2 26621.255} C_VEL
LIN {X 0,Y 221.678,Z 1227.589,A -85,B 0,C 180,E1 26628.197,E2 26628.197} C_VEL
LIN {X 0,Y 211.785,Z 1224.588,A -85,B 0,C 180,E1 26635.927,E2 26635.927} C_VEL
LIN {X 0,Y 205.61,Z 1215.982,A -85,B 0,C 180,E1 26645.138,E2 26645.138} C_VEL
LIN {X 0,Y 204.371,Z 1201.92,A -85,B 0,C 180,E1 26654.168,E2 26654.168} C_VEL
LIN {X 0,Y 206.181,Z 1183.168,A -85,B 0,C 180,E1 26662.202,E2 26662.202} C_VEL
LIN {X 0,Y 210.309,Z 1158.553,A -85,B 0,C 180,E1 26669.426,E2 26669.426} C_VEL
LIN {X 0,Y 215.361,Z 1130.669,A -85,B 0,C 180,E1 26675.026,E2 26675.026} C_VEL
LIN {X 0,Y 220.452,Z 1098.855,A -85,B 0,C 180,E1 26679.214,E2 26679.214} C_VEL
LIN {X 0,Y 223.722,Z 1066.188,A -85,B 0,C 180,E1 26682.138,E2 26682.138} C_VEL
LIN {X 0,Y 221.846,Z 1057.929,A -85,B 0,C 180,E1 26683.062,E2 26683.062} C_VEL
LIN {X 0,Y 216.811,Z 1047.206,A -85,B 0,C 180,E1 26684.548,E2 26684.548} C_VEL
LIN {X 0,Y 207.583,Z 1032.096,A -85,B 0,C 180,E1 26687.017,E2 26687.017} C_VEL
LIN {X 0,Y 206.99,Z 1030.181,A -85,B 0,C 180,E1 26687.273,E2 26687.273} C_VEL
LIN {X 0,Y 193.719,Z 989.336,A -85,B 0,C 180,E1 26693.024,E2 26693.024} C_VEL
LIN {X 0,Y 189.634,Z 977.53,A -85,B 0,C 180,E1 26694.931,E2 26694.931} C_VEL
LIN {X 0,Y 190.394,Z 977.53,A -85,B 0,C 180,E1 26706.528,E2 26706.528} C_VEL
LIN {X 0,Y 191.334,Z 977.53,A -85,B 0,C 180,E1 26716.234,E2 26716.234} C_VEL
LIN {X 0,Y 192.584,Z 977.53,A -85,B 0,C 180,E1 26725.466,E2 26725.466} C_VEL
LIN {X 0,Y 193.265,Z 977.53,A -85,B 0,C 180,E1 26729.979,E2 26729.979} C_VEL
LIN {X 0,Y 191.948,Z 977.53,A -85,B 0,C 180,E1 26739.063,E2 26739.063} C_VEL
LIN {X 0,Y 190.778,Z 977.863,A -85,B 0,C 180,E1 26749.655,E2 26749.655} C_VEL
LIN {X 0,Y 211.005,Z 1024.672,A -85,B 0,C 180,E1 26758.387,E2 26758.387} C_VEL
LIN {X 0,Y 223.783,Z 1061.676,A -85,B 0,C 180,E1 26764.231,E2 26764.231} C_VEL
LIN {X 0,Y 233.479,Z 1098.421,A -85,B 0,C 180,E1 26770.108,E2 26770.108} C_VEL
LIN {X 0,Y 235.595,Z 1108.991,A -85,B 0,C 180,E1 26771.848,E2 26771.848} C_VEL
LIN {X 0,Y 223.688,Z 1148.623,A -85,B 0,C 180,E1 26777.328,E2 26777.328} C_VEL
LIN {X 0,Y 212.397,Z 1182.768,A -85,B 0,C 180,E1 26784.229,E2 26784.229} C_VEL
LIN {X 0,Y 203.419,Z 1210.719,A -85,B 0,C 180,E1 26792.223,E2 26792.223} C_VEL
LIN {X 0,Y 197.293,Z 1233.866,A -85,B 0,C 180,E1 26801.499,E2 26801.499} C_VEL
LIN {X 0,Y 194.55,Z 1250.827,A -85,B 0,C 180,E1 26811.007,E2 26811.007} C_VEL
LIN {X 0,Y 194.07,Z 1263.313,A -85,B 0,C 180,E1 26821.086,E2 26821.086} C_VEL
LIN {X 0,Y 196.773,Z 1272.581,A -85,B 0,C 180,E1 26833.323,E2 26833.323} C_VEL
LIN {X 0,Y 207.409,Z 1276.979,A -85,B 0,C 180,E1 26845.961,E2 26845.961} C_VEL
LIN {X 0,Y 227.083,Z 1276.519,A -85,B 0,C 180,E1 26856.87,E2 26856.87} C_VEL
LIN {X 0,Y 244.713,Z 1273.847,A -85,B 0,C 180,E1 26862.89,E2 26862.89} C_VEL
LIN {X 0,Y 213.169,Z 1283.345,A -85,B 0,C 180,E1 26875.366,E2 26875.366} C_VEL
LIN {X 0,Y 198.879,Z 1286.25,A -85,B 0,C 180,E1 26887.629,E2 26887.629} C_VEL
LIN {X 0,Y 194.362,Z 1283.819,A -85,B 0,C 180,E1 26901.051,E2 26901.051} C_VEL
LIN {X 0,Y 195.257,Z 1278.429,A -85,B 0,C 180,E1 26910.021,E2 26910.021} C_VEL
LIN {X 0,Y 195.28,Z 1269.982,A -85,B 0,C 180,E1 26917.825,E2 26917.825} C_VEL
LIN {X 0,Y 196.144,Z 1258.944,A -85,B 0,C 180,E1 26925.283,E2 26925.283} C_VEL
LIN {X 0,Y 201.163,Z 1255.87,A -85,B 0,C 180,E1 26936.891,E2 26936.891} C_VEL
LIN {X 0,Y 217.127,Z 1246.856,A -85,B 0,C 180,E1 26948.933,E2 26948.933} C_VEL
LIN {X 0,Y 242.513,Z 1232.171,A -85,B 0,C 180,E1 26958.596,E2 26958.596} C_VEL
LIN {X 0,Y 274.821,Z 1211.718,A -85,B 0,C 180,E1 26965.822,E2 26965.822} C_VEL
LIN {X 0,Y 278.734,Z 1209.047,A -85,B 0,C 180,E1 26966.463,E2 26966.463} C_VEL
LIN {X 0,Y 278.094,Z 1209.243,A -85,B 0,C 180,E1 26967.015,E2 26967.015} C_VEL
LIN {X 0,Y 253.082,Z 1221.089,A -85,B 0,C 180,E1 26972.385,E2 26972.385} C_VEL
LIN {X 0,Y 236.386,Z 1226.529,A -85,B 0,C 180,E1 26977.412,E2 26977.412} C_VEL
LIN {X 0,Y 220.475,Z 1228.96,A -85,B 0,C 180,E1 26984.075,E2 26984.075} C_VEL
LIN {X 0,Y 208.325,Z 1227.336,A -85,B 0,C 180,E1 26991.667,E2 26991.667} C_VEL
LIN {X 0,Y 199.592,Z 1220.316,A -85,B 0,C 180,E1 27001.118,E2 27001.118} C_VEL
LIN {X 0,Y 196.485,Z 1208.873,A -85,B 0,C 180,E1 27010.023,E2 27010.023} C_VEL
LIN {X 0,Y 197.151,Z 1192.652,A -85,B 0,C 180,E1 27018.515,E2 27018.515} C_VEL
LIN {X 0,Y 200.293,Z 1170.27,A -85,B 0,C 180,E1 27026.529,E2 27026.529} C_VEL
LIN {X 0,Y 205.245,Z 1143.879,A -85,B 0,C 180,E1 27033.02,E2 27033.02} C_VEL
LIN {X 0,Y 210.657,Z 1113.028,A -85,B 0,C 180,E1 27038.128,E2 27038.128} C_VEL
LIN {X 0,Y 215.622,Z 1077.519,A -85,B 0,C 180,E1 27041.802,E2 27041.802} C_VEL
LIN {X 0,Y 215.968,Z 1066.598,A -85,B 0,C 180,E1 27042.823,E2 27042.823} C_VEL
LIN {X 0,Y 206.99,Z 1030.181,A -85,B 0,C 180,E1 27047.273,E2 27047.273} C_VEL
LIN {X 0,Y 201.736,Z 1019.761,A -85,B 0,C 180,E1 27048.948,E2 27048.948} C_VEL
LIN {X 0,Y 190.968,Z 1003.663,A -85,B 0,C 180,E1 27052.096,E2 27052.096} C_VEL
LIN {X 0,Y 181.657,Z 977.53,A -85,B 0,C 180,E1 27056.578,E2 27056.578} C_VEL
LIN {X 0,Y 182.393,Z 977.53,A -85,B 0,C 180,E1 27066.111,E2 27066.111} C_VEL
LIN {X 0,Y 183.314,Z 977.53,A -85,B 0,C 180,E1 27075.619,E2 27075.619} C_VEL
LIN {X 0,Y 184.611,Z 977.53,A -85,B 0,C 180,E1 27085.27,E2 27085.27} C_VEL
LIN {X 0,Y 185.337,Z 977.53,A -85,B 0,C 180,E1 27089.978,E2 27089.978} C_VEL
LIN {X 0,Y 183.947,Z 977.53,A -85,B 0,C 180,E1 27099.46,E2 27099.46} C_VEL
LIN {X 0,Y 183.099,Z 977.715,A -85,B 0,C 180,E1 27107.509,E2 27107.509} C_VEL
LIN {X 0,Y 202.436,Z 1022.562,A -85,B 0,C 180,E1 27116.499,E2 27116.499} C_VEL
LIN {X 0,Y 215.053,Z 1058.504,A -85,B 0,C 180,E1 27122.49,E2 27122.49} C_VEL
LIN {X 0,Y 225.281,Z 1096.211,A -85,B 0,C 180,E1 27128.773,E2 27128.773} C_VEL
LIN {X 0,Y 227.98,Z 1110.581,A -85,B 0,C 180,E1 27131.196,E2 27131.196} C_VEL
LIN {X 0,Y 215.533,Z 1150.729,A -85,B 0,C 180,E1 27137.011,E2 27137.011} C_VEL
LIN {X 0,Y 204.133,Z 1184.393,A -85,B 0,C 180,E1 27144.145,E2 27144.145} C_VEL
LIN {X 0,Y 194.756,Z 1213.172,A -85,B 0,C 180,E1 27152.876,E2 27152.876} C_VEL
LIN {X 0,Y 188.728,Z 1236.837,A -85,B 0,C 180,E1 27163.113,E2 27163.113} C_VEL
LIN {X 0,Y 186.397,Z 1252.91,A -85,B 0,C 180,E1 27172.963,E2 27172.963} C_VEL
LIN {X 0,Y 186.356,Z 1264.732,A -85,B 0,C 180,E1 27183.462,E2 27183.462} C_VEL
LIN {X 0,Y 190.269,Z 1273.538,A -85,B 0,C 180,E1 27196.149,E2 27196.149} C_VEL
LIN {X 0,Y 200.32,Z 1277.38,A -85,B 0,C 180,E1 27206.953,E2 27206.953} C_VEL
LIN {X 0,Y 220.855,Z 1277.599,A -85,B 0,C 180,E1 27218.091,E2 27218.091} C_VEL
LIN {X 0,Y 233.747,Z 1276.279,A -85,B 0,C 180,E1 27222.572,E2 27222.572} C_VEL
LIN {X 0,Y 233.223,Z 1276.591,A -85,B 0,C 180,E1 27223.404,E2 27223.404} C_VEL
LIN {X 0,Y 206.628,Z 1283.32,A -85,B 0,C 180,E1 27234.104,E2 27234.104} C_VEL
LIN {X 0,Y 191.513,Z 1285.501,A -85,B 0,C 180,E1 27246.719,E2 27246.719} C_VEL
LIN {X 0,Y 186.605,Z 1282.564,A -85,B 0,C 180,E1 27260.676,E2 27260.676} C_VEL
LIN {X 0,Y 187.532,Z 1276.829,A -85,B 0,C 180,E1 27270.022,E2 27270.022} C_VEL
LIN {X 0,Y 187.518,Z 1268.024,A -85,B 0,C 180,E1 27278.151,E2 27278.151} C_VEL
LIN {X 0,Y 188.374,Z 1257.558,A -85,B 0,C 180,E1 27285.295,E2 27285.295} C_VEL
LIN {X 0,Y 193.975,Z 1254.981,A -85,B 0,C 180,E1 27297.973,E2 27297.973} C_VEL
LIN {X 0,Y 210.907,Z 1246.627,A -85,B 0,C 180,E1 27310.311,E2 27310.311} C_VEL
LIN {X 0,Y 237.352,Z 1232.914,A -85,B 0,C 180,E1 27320.03,E2 27320.03} C_VEL
LIN {X 0,Y 266.096,Z 1216.357,A -85,B 0,C 180,E1 27326.409,E2 27326.409} C_VEL
LIN {X 0,Y 267.125,Z 1215.592,A -85,B 0,C 180,E1 27326.991,E2 27326.991} C_VEL
LIN {X 0,Y 243.66,Z 1224.877,A -85,B 0,C 180,E1 27332.231,E2 27332.231} C_VEL
LIN {X 0,Y 220.559,Z 1229.965,A -85,B 0,C 180,E1 27339.942,E2 27339.942} C_VEL
LIN {X 0,Y 206.14,Z 1229.61,A -85,B 0,C 180,E1 27347.293,E2 27347.293} C_VEL
LIN {X 0,Y 195.806,Z 1225.125,A -85,B 0,C 180,E1 27355.594,E2 27355.594} C_VEL
LIN {X 0,Y 189.507,Z 1214.651,A -85,B 0,C 180,E1 27365.768,E2 27365.768} C_VEL
LIN {X 0,Y 188.722,Z 1198.128,A -85,B 0,C 180,E1 27375.868,E2 27375.868} C_VEL
LIN {X 0,Y 191.142,Z 1178.115,A -85,B 0,C 180,E1 27384.162,E2 27384.162} C_VEL
LIN {X 0,Y 195.747,Z 1152.173,A -85,B 0,C 180,E1 27391.585,E2 27391.585} C_VEL
LIN {X 0,Y 201.26,Z 1122.685,A -85,B 0,C 180,E1 27397.278,E2 27397.278} C_VEL
LIN {X 0,Y 206.571,Z 1089.881,A -85,B 0,C 180,E1 27401.348,E2 27401.348} C_VEL
LIN {X 0,Y 208.569,Z 1068.501,A -85,B 0,C 180,E1 27403.378,E2 27403.378} C_VEL
LIN {X 0,Y 196.894,Z 1022.238,A -85,B 0,C 180,E1 27409.368,E2 27409.368} C_VEL
LIN {X 0,Y 190.968,Z 1003.663,A -85,B 0,C 180,E1 27412.096,E2 27412.096} C_VEL
LIN {X 0,Y 184.228,Z 996.146,A -85,B 0,C 180,E1 27413.99,E2 27413.99} C_VEL
LIN {X 0,Y 177.592,Z 988.608,A -85,B 0,C 180,E1 27415.984,E2 27415.984} C_VEL
LIN {X 0,Y 173.734,Z 977.53,A -85,B 0,C 180,E1 27417.979,E2 27417.979} C_VEL
LIN {X 0,Y 174.674,Z 977.53,A -85,B 0,C 180,E1 27429.672,E2 27429.672} C_VEL
LIN {X 0,Y 175.937,Z 977.53,A -85,B 0,C 180,E1 27440.058,E2 27440.058} C_VEL
LIN {X 0,Y 177.422,Z 977.53,A -85,B 0,C 180,E1 27449.977,E2 27449.977} C_VEL
LIN {X 0,Y 175.911,Z 977.53,A -85,B 0,C 180,E1 27459.897,E2 27459.897} C_VEL
LIN {X 0,Y 175.289,Z 977.951,A -85,B 0,C 180,E1 27465.165,E2 27465.165} C_VEL
LIN {X 0,Y 194.034,Z 1020.491,A -85,B 0,C 180,E1 27474.488,E2 27474.488} C_VEL
LIN {X 0,Y 206.81,Z 1056.393,A -85,B 0,C 180,E1 27480.833,E2 27480.833} C_VEL
LIN {X 0,Y 217.023,Z 1093.839,A -85,B 0,C 180,E1 27487.318,E2 27487.318} C_VEL
LIN {X 0,Y 220.526,Z 1111.622,A -85,B 0,C 180,E1 27490.467,E2 27490.467} C_VEL
LIN {X 0,Y 207.779,Z 1151.605,A -85,B 0,C 180,E1 27496.457,E2 27496.457} C_VEL
LIN {X 0,Y 196.006,Z 1185.46,A -85,B 0,C 180,E1 27503.94,E2 27503.94} C_VEL
LIN {X 0,Y 186.722,Z 1213.642,A -85,B 0,C 180,E1 27512.887,E2 27512.887} C_VEL
LIN {X 0,Y 180.892,Z 1236,A -85,B 0,C 180,E1 27522.918,E2 27522.918} C_VEL
LIN {X 0,Y 178.467,Z 1253.263,A -85,B 0,C 180,E1 27533.874,E2 27533.874} C_VEL
LIN {X 0,Y 178.51,Z 1264,A -85,B 0,C 180,E1 27543.615,E2 27543.615} C_VEL
LIN {X 0,Y 182.628,Z 1273.332,A -85,B 0,C 180,E1 27556.771,E2 27556.771} C_VEL
LIN {X 0,Y 199.427,Z 1278.474,A -85,B 0,C 180,E1 27572.091,E2 27572.091} C_VEL
LIN {X 0,Y 223.801,Z 1278.114,A -85,B 0,C 180,E1 27582.57,E2 27582.57} C_VEL
LIN {X 0,Y 207.809,Z 1281.721,A -85,B 0,C 180,E1 27589.012,E2 27589.012} C_VEL
LIN {X 0,Y 186.02,Z 1284.783,A -85,B 0,C 180,E1 27603.552,E2 27603.552} C_VEL
LIN {X 0,Y 179.563,Z 1283.064,A -85,B 0,C 180,E1 27615.359,E2 27615.359} C_VEL
LIN {X 0,Y 179.366,Z 1277.087,A -85,B 0,C 180,E1 27627.602,E2 27627.602} C_VEL
LIN {X 0,Y 179.786,Z 1270.466,A -85,B 0,C 180,E1 27634.857,E2 27634.857} C_VEL
LIN {X 0,Y 180.639,Z 1256.041,A -85,B 0,C 180,E1 27645.281,E2 27645.281} C_VEL
LIN {X 0,Y 186.873,Z 1253.976,A -85,B 0,C 180,E1 27659.136,E2 27659.136} C_VEL
LIN {X 0,Y 204.825,Z 1246.369,A -85,B 0,C 180,E1 27671.771,E2 27671.771} C_VEL
LIN {X 0,Y 232.348,Z 1233.56,A -85,B 0,C 180,E1 27681.525,E2 27681.525} C_VEL
LIN {X 0,Y 255.945,Z 1221.209,A -85,B 0,C 180,E1 27686.987,E2 27686.987} C_VEL
LIN {X 0,Y 231.627,Z 1228.838,A -85,B 0,C 180,E1 27692.78,E2 27692.78} C_VEL
LIN {X 0,Y 213.167,Z 1231.567,A -85,B 0,C 180,E1 27699.215,E2 27699.215} C_VEL
LIN {X 0,Y 195.312,Z 1229.532,A -85,B 0,C 180,E1 27708.85,E2 27708.85} C_VEL
LIN {X 0,Y 185.003,Z 1222.095,A -85,B 0,C 180,E1 27718.86,E2 27718.86} C_VEL
LIN {X 0,Y 180.724,Z 1208.58,A -85,B 0,C 180,E1 27729.687,E2 27729.687} C_VEL
LIN {X 0,Y 181.376,Z 1191.967,A -85,B 0,C 180,E1 27738.67,E2 27738.67} C_VEL
LIN {X 0,Y 184.773,Z 1168.97,A -85,B 0,C 180,E1 27747.306,E2 27747.306} C_VEL
LIN {X 0,Y 190.125,Z 1141.68,A -85,B 0,C 180,E1 27754.289,E2 27754.289} C_VEL
LIN {X 0,Y 195.609,Z 1111.79,A -85,B 0,C 180,E1 27759.437,E2 27759.437} C_VEL
LIN {X 0,Y 201.375,Z 1072.062,A -85,B 0,C 180,E1 27763.727,E2 27763.727} C_VEL
LIN {X 0,Y 190.606,Z 1027.471,A -85,B 0,C 180,E1 27769.738,E2 27769.738} C_VEL
LIN {X 0,Y 177.592,Z 988.608,A -85,B 0,C 180,E1 27775.984,E2 27775.984} C_VEL
LIN {X 0,Y 173.227,Z 981.881,A -85,B 0,C 180,E1 27778.241,E2 27778.241} C_VEL
LIN {X 0,Y 167.386,Z 977.969,A -85,B 0,C 180,E1 27782.832,E2 27782.832} C_VEL
LIN {X 0,Y 166.206,Z 977.53,A -85,B 0,C 180,E1 27785.859,E2 27785.859} C_VEL
LIN {X 0,Y 167.2,Z 977.53,A -85,B 0,C 180,E1 27794.199,E2 27794.199} C_VEL
LIN {X 0,Y 168.65,Z 977.53,A -85,B 0,C 180,E1 27804.821,E2 27804.821} C_VEL
LIN {X 0,Y 169.488,Z 977.53,A -85,B 0,C 180,E1 27809.976,E2 27809.976} C_VEL
LIN {X 0,Y 167.903,Z 977.53,A -85,B 0,C 180,E1 27820.374,E2 27820.374} C_VEL
LIN {X 0,Y 167.521,Z 977.841,A -85,B 0,C 180,E1 27822.546,E2 27822.546} C_VEL
LIN {X 0,Y 184.342,Z 1015.523,A -85,B 0,C 180,E1 27831.708,E2 27831.708} C_VEL
LIN {X 0,Y 197.27,Z 1050.275,A -85,B 0,C 180,E1 27838.354,E2 27838.354} C_VEL
LIN {X 0,Y 207.346,Z 1086.011,A -85,B 0,C 180,E1 27844.791,E2 27844.791} C_VEL
LIN {X 0,Y 212.913,Z 1113.194,A -85,B 0,C 180,E1 27849.766,E2 27849.766} C_VEL
LIN {X 0,Y 199.993,Z 1152.445,A -85,B 0,C 180,E1 27855.88,E2 27855.88} C_VEL
LIN {X 0,Y 187.948,Z 1186.334,A -85,B 0,C 180,E1 27863.691,E2 27863.691} C_VEL
LIN {X 0,Y 178.275,Z 1215.447,A -85,B 0,C 180,E1 27873.447,E2 27873.447} C_VEL
LIN {X 0,Y 172.449,Z 1238.595,A -85,B 0,C 180,E1 27884.681,E2 27884.681} C_VEL
LIN {X 0,Y 170.542,Z 1253.549,A -85,B 0,C 180,E1 27894.867,E2 27894.867} C_VEL
LIN {X 0,Y 170.781,Z 1264.267,A -85,B 0,C 180,E1 27905.053,E2 27905.053} C_VEL
LIN {X 0,Y 176.805,Z 1274.283,A -85,B 0,C 180,E1 27920.008,E2 27920.008} C_VEL
LIN {X 0,Y 192.779,Z 1278.951,A -85,B 0,C 180,E1 27933.338,E2 27933.338} C_VEL
LIN {X 0,Y 213.214,Z 1279.487,A -85,B 0,C 180,E1 27942.344,E2 27942.344} C_VEL
LIN {X 0,Y 210.779,Z 1280.173,A -85,B 0,C 180,E1 27944.065,E2 27944.065} C_VEL
LIN {X 0,Y 187.056,Z 1283.696,A -85,B 0,C 180,E1 27955.482,E2 27955.482} C_VEL
LIN {X 0,Y 173.777,Z 1283.191,A -85,B 0,C 180,E1 27969.612,E2 27969.612} C_VEL
LIN {X 0,Y 171.068,Z 1278.571,A -85,B 0,C 180,E1 27982.389,E2 27982.389} C_VEL
LIN {X 0,Y 172.052,Z 1272.345,A -85,B 0,C 180,E1 27991.285,E2 27991.285} C_VEL
LIN {X 0,Y 172.136,Z 1262.178,A -85,B 0,C 180,E1 28000.164,E2 28000.164} C_VEL
LIN {X 0,Y 172.933,Z 1254.387,A -85,B 0,C 180,E1 28005.614,E2 28005.614} C_VEL
LIN {X 0,Y 179.87,Z 1252.921,A -85,B 0,C 180,E1 28020.387,E2 28020.387} C_VEL
LIN {X 0,Y 198.907,Z 1246.043,A -85,B 0,C 180,E1 28033.312,E2 28033.312} C_VEL
LIN {X 0,Y 229.402,Z 1233.248,A -85,B 0,C 180,E1 28043.563,E2 28043.563} C_VEL
LIN {X 0,Y 242.868,Z 1227,A -85,B 0,C 180,E1 28046.538,E2 28046.538} C_VEL
LIN {X 0,Y 243.838,Z 1226.342,A -85,B 0,C 180,E1 28047.174,E2 28047.174} C_VEL
LIN {X 0,Y 221.391,Z 1231.675,A -85,B 0,C 180,E1 28052.882,E2 28052.882} C_VEL
LIN {X 0,Y 205.779,Z 1233.035,A -85,B 0,C 180,E1 28058.432,E2 28058.432} C_VEL
LIN {X 0,Y 187.451,Z 1230.006,A -85,B 0,C 180,E1 28068.376,E2 28068.376} C_VEL
LIN {X 0,Y 176.988,Z 1221.726,A -85,B 0,C 180,E1 28078.809,E2 28078.809} C_VEL
LIN {X 0,Y 172.786,Z 1207.359,A -85,B 0,C 180,E1 28090.137,E2 28090.137} C_VEL
LIN {X 0,Y 173.939,Z 1187.824,A -85,B 0,C 180,E1 28100.428,E2 28100.428} C_VEL
LIN {X 0,Y 177.772,Z 1163.933,A -85,B 0,C 180,E1 28109.034,E2 28109.034} C_VEL
LIN {X 0,Y 183.246,Z 1136.722,A -85,B 0,C 180,E1 28115.769,E2 28115.769} C_VEL
LIN {X 0,Y 189.349,Z 1103.799,A -85,B 0,C 180,E1 28121.119,E2 28121.119} C_VEL
LIN {X 0,Y 193.393,Z 1070.607,A -85,B 0,C 180,E1 28124.731,E2 28124.731} C_VEL
LIN {X 0,Y 182.52,Z 1026.266,A -85,B 0,C 180,E1 28131.081,E2 28131.081} C_VEL
LIN {X 0,Y 169.153,Z 986.808,A -85,B 0,C 180,E1 28137.909,E2 28137.909} C_VEL
LIN {X 0,Y 165.878,Z 977.53,A -85,B 0,C 180,E1 28139.863,E2 28139.863} C_VEL
LIN {X 0,Y 166.206,Z 977.53,A -85,B 0,C 180,E1 28145.859,E2 28145.859} C_VEL
LIN {X 0,Y 163.937,Z 977.53,A -85,B 0,C 180,E1 28150.349,E2 28150.349} C_VEL
LIN {X 0,Y 159.591,Z 977.53,A -85,B 0,C 180,E1 28158.082,E2 28158.082} C_VEL
LIN {X 0,Y 160.676,Z 977.53,A -85,B 0,C 180,E1 28164.563,E2 28164.563} C_VEL
LIN {X 0,Y 161.569,Z 977.53,A -85,B 0,C 180,E1 28169.975,E2 28169.975} C_VEL
LIN {X 0,Y 160.059,Z 977.871,A -85,B 0,C 180,E1 28179.762,E2 28179.762} C_VEL
LIN {X 0,Y 175.953,Z 1013.506,A -85,B 0,C 180,E1 28189.28,E2 28189.28} C_VEL
LIN {X 0,Y 189.1,Z 1048.365,A -85,B 0,C 180,E1 28196.446,E2 28196.446} C_VEL
LIN {X 0,Y 199.558,Z 1085.223,A -85,B 0,C 180,E1 28203.43,E2 28203.43} C_VEL
LIN {X 0,Y 205.527,Z 1113.883,A -85,B 0,C 180,E1 28208.915,E2 28208.915} C_VEL
LIN {X 0,Y 192.085,Z 1153.578,A -85,B 0,C 180,E1 28215.339,E2 28215.339} C_VEL
LIN {X 0,Y 179.988,Z 1186.874,A -85,B 0,C 180,E1 28223.347,E2 28223.347} C_VEL
LIN {X 0,Y 170.208,Z 1215.878,A -85,B 0,C 180,E1 28233.532,E2 28233.532} C_VEL
LIN {X 0,Y 164.368,Z 1238.976,A -85,B 0,C 180,E1 28245.329,E2 28245.329} C_VEL
LIN {X 0,Y 162.642,Z 1255.378,A -85,B 0,C 180,E1 28257.292,E2 28257.292} C_VEL
LIN {X 0,Y 163.382,Z 1265.502,A -85,B 0,C 180,E1 28267.957,E2 28267.957} C_VEL
LIN {X 0,Y 171.391,Z 1275.146,A -85,B 0,C 180,E1 28283.401,E2 28283.401} C_VEL
LIN {X 0,Y 195.05,Z 1280.068,A -85,B 0,C 180,E1 28299.059,E2 28299.059} C_VEL
LIN {X 0,Y 202.842,Z 1280.372,A -85,B 0,C 180,E1 28302.198,E2 28302.198} C_VEL
LIN {X 0,Y 203.456,Z 1280.533,A -85,B 0,C 180,E1 28303.113,E2 28303.113} C_VEL
LIN {X 0,Y 180.518,Z 1283.166,A -85,B 0,C 180,E1 28314.042,E2 28314.042} C_VEL
LIN {X 0,Y 166.369,Z 1281.982,A -85,B 0,C 180,E1 28328.661,E2 28328.661} C_VEL
LIN {X 0,Y 163.368,Z 1277.033,A -85,B 0,C 180,E1 28342.028,E2 28342.028} C_VEL
LIN {X 0,Y 164.367,Z 1270.469,A -85,B 0,C 180,E1 28351.345,E2 28351.345} C_VEL
LIN {X 0,Y 164.54,Z 1258.2,A -85,B 0,C 180,E1 28361.892,E2 28361.892} C_VEL
LIN {X 0,Y 165.253,Z 1252.633,A -85,B 0,C 180,E1 28365.992,E2 28365.992} C_VEL
LIN {X 0,Y 172.958,Z 1251.783,A -85,B 0,C 180,E1 28381.74,E2 28381.74} C_VEL
LIN {X 0,Y 194.396,Z 1245.164,A -85,B 0,C 180,E1 28395.502,E2 28395.502} C_VEL
LIN {X 0,Y 222.844,Z 1234.568,A -85,B 0,C 180,E1 28404.714,E2 28404.714} C_VEL
LIN {X 0,Y 231.353,Z 1231.054,A -85,B 0,C 180,E1 28406.668,E2 28406.668} C_VEL
LIN {X 0,Y 232.409,Z 1230.462,A -85,B 0,C 180,E1 28407.23,E2 28407.23} C_VEL
LIN {X 0,Y 207.716,Z 1234.229,A -85,B 0,C 180,E1 28414.08,E2 28414.08} C_VEL
LIN {X 0,Y 190.112,Z 1233.448,A -85,B 0,C 180,E1 28421.445,E2 28421.445} C_VEL
LIN {X 0,Y 174.077,Z 1226.951,A -85,B 0,C 180,E1 28432.534,E2 28432.534} C_VEL
LIN {X 0,Y 166.191,Z 1214.737,A -85,B 0,C 180,E1 28444.38,E2 28444.38} C_VEL
LIN {X 0,Y 165.097,Z 1196.652,A -85,B 0,C 180,E1 28456.019,E2 28456.019} C_VEL
LIN {X 0,Y 168.117,Z 1173.926,A -85,B 0,C 180,E1 28465.935,E2 28465.935} C_VEL
LIN {X 0,Y 173.585,Z 1146.123,A -85,B 0,C 180,E1 28474.131,E2 28474.131} C_VEL
LIN {X 0,Y 179.534,Z 1116.125,A -85,B 0,C 180,E1 28480.015,E2 28480.015} C_VEL
LIN {X 0,Y 185.745,Z 1077.823,A -85,B 0,C 180,E1 28484.738,E2 28484.738} C_VEL
LIN {X 0,Y 185.033,Z 1067.805,A -85,B 0,C 180,E1 28486.01,E2 28486.01} C_VEL
LIN {X 0,Y 173.958,Z 1023.49,A -85,B 0,C 180,E1 28492.793,E2 28492.793} C_VEL
LIN {X 0,Y 160.948,Z 986.086,A -85,B 0,C 180,E1 28499.805,E2 28499.805} C_VEL
LIN {X 0,Y 158.066,Z 977.53,A -85,B 0,C 180,E1 28501.73,E2 28501.73} C_VEL
LIN {X 0,Y 159.077,Z 977.53,A -85,B 0,C 180,E1 28513.369,E2 28513.369} C_VEL
LIN {X 0,Y 159.591,Z 977.53,A -85,B 0,C 180,E1 28518.082,E2 28518.082} C_VEL
LIN {X 0,Y 158.329,Z 977.53,A -85,B 0,C 180,E1 28522.773,E2 28522.773} C_VEL
LIN {X 0,Y 153.39,Z 977.53,A -85,B 0,C 180,E1 28530.809,E2 28530.809} C_VEL
LIN {X 0,Y 152.534,Z 977.53,A -85,B 0,C 180,E1 28536.496,E2 28536.496} C_VEL
LIN {X 0,Y 154.705,Z 983.235,A -85,B 0,C 180,E1 28538.308,E2 28538.308} C_VEL
LIN {X 0,Y 168.547,Z 1013.588,A -85,B 0,C 180,E1 28547.132,E2 28547.132} C_VEL
LIN {X 0,Y 180.991,Z 1046.37,A -85,B 0,C 180,E1 28554.371,E2 28554.371} C_VEL
LIN {X 0,Y 191.343,Z 1082.629,A -85,B 0,C 180,E1 28561.619,E2 28561.619} C_VEL
LIN {X 0,Y 198.065,Z 1113.885,A -85,B 0,C 180,E1 28567.901,E2 28567.901} C_VEL
LIN {X 0,Y 185.514,Z 1151.256,A -85,B 0,C 180,E1 28574.063,E2 28574.063} C_VEL
LIN {X 0,Y 172.672,Z 1185.571,A -85,B 0,C 180,E1 28582.458,E2 28582.458} C_VEL
LIN {X 0,Y 162.578,Z 1214.601,A -85,B 0,C 180,E1 28592.937,E2 28592.937} C_VEL
LIN {X 0,Y 156.464,Z 1238.41,A -85,B 0,C 180,E1 28605.464,E2 28605.464} C_VEL
LIN {X 0,Y 154.834,Z 1253.94,A -85,B 0,C 180,E1 28617.156,E2 28617.156} C_VEL
LIN {X 0,Y 155.625,Z 1264.572,A -85,B 0,C 180,E1 28628.357,E2 28628.357} C_VEL
LIN {X 0,Y 164.164,Z 1274.802,A -85,B 0,C 180,E1 28644.497,E2 28644.497} C_VEL
LIN {X 0,Y 187.936,Z 1280.491,A -85,B 0,C 180,E1 28660.118,E2 28660.118} C_VEL
LIN {X 0,Y 193.019,Z 1280.822,A -85,B 0,C 180,E1 28662.221,E2 28662.221} C_VEL
LIN {X 0,Y 193.511,Z 1281.001,A -85,B 0,C 180,E1 28663.079,E2 28663.079} C_VEL
LIN {X 0,Y 167.741,Z 1282.391,A -85,B 0,C 180,E1 28677.209,E2 28677.209} C_VEL
LIN {X 0,Y 156.794,Z 1279.096,A -85,B 0,C 180,E1 28693.174,E2 28693.174} C_VEL
LIN {X 0,Y 156.295,Z 1271.894,A -85,B 0,C 180,E1 28707.247,E2 28707.247} C_VEL
LIN {X 0,Y 156.608,Z 1264.317,A -85,B 0,C 180,E1 28715.578,E2 28715.578} C_VEL
LIN {X 0,Y 157.593,Z 1250.732,A -85,B 0,C 180,E1 28726.115,E2 28726.115} C_VEL
LIN {X 0,Y 166.174,Z 1250.526,A -85,B 0,C 180,E1 28743.198,E2 28743.198} C_VEL
LIN {X 0,Y 187.527,Z 1245.071,A -85,B 0,C 180,E1 28756.685,E2 28756.685} C_VEL
LIN {X 0,Y 218.357,Z 1234.945,A -85,B 0,C 180,E1 28766.413,E2 28766.413} C_VEL
LIN {X 0,Y 220.579,Z 1233.943,A -85,B 0,C 180,E1 28767.37,E2 28767.37} C_VEL
LIN {X 0,Y 200.621,Z 1235.76,A -85,B 0,C 180,E1 28773.091,E2 28773.091} C_VEL
LIN {X 0,Y 178.689,Z 1233.215,A -85,B 0,C 180,E1 28782.773,E2 28782.773} C_VEL
LIN {X 0,Y 164.951,Z 1225.649,A -85,B 0,C 180,E1 28793.445,E2 28793.445} C_VEL
LIN {X 0,Y 157.877,Z 1212.374,A -85,B 0,C 180,E1 28805.546,E2 28805.546} C_VEL
LIN {X 0,Y 157.312,Z 1194.514,A -85,B 0,C 180,E1 28816.835,E2 28816.835} C_VEL
LIN {X 0,Y 160.52,Z 1171.993,A -85,B 0,C 180,E1 28826.7,E2 28826.7} C_VEL
LIN {X 0,Y 165.845,Z 1145.758,A -85,B 0,C 180,E1 28834.642,E2 28834.642} C_VEL
LIN {X 0,Y 172.397,Z 1113.481,A -85,B 0,C 180,E1 28841.096,E2 28841.096} C_VEL
LIN {X 0,Y 178.584,Z 1074.317,A -85,B 0,C 180,E1 28845.983,E2 28845.983} C_VEL
LIN {X 0,Y 168.172,Z 1030.138,A -85,B 0,C 180,E1 28853.018,E2 28853.018} C_VEL
LIN {X 0,Y 156.029,Z 993.638,A -85,B 0,C 180,E1 28860.062,E2 28860.062} C_VEL
LIN {X 0,Y 150.235,Z 977.53,A -85,B 0,C 180,E1 28863.867,E2 28863.867} C_VEL
LIN {X 0,Y 151.004,Z 977.53,A -85,B 0,C 180,E1 28872.452,E2 28872.452} C_VEL
LIN {X 0,Y 152.658,Z 977.53,A -85,B 0,C 180,E1 28884.277,E2 28884.277} C_VEL
LIN {X 0,Y 153.39,Z 977.53,A -85,B 0,C 180,E1 28890.809,E2 28890.809} C_VEL
LIN {X 0,Y 152.612,Z 980.543,A -85,B 0,C 180,E1 28894.199,E2 28894.199} C_VEL
LIN {X 0,Y 153.044,Z 992.58,A -85,B 0,C 180,E1 28898.676,E2 28898.676} C_VEL
LIN {X 0,Y 155.053,Z 999.711,A -85,B 0,C 180,E1 28900.778,E2 28900.778} C_VEL
LIN {X 0,Y 168.533,Z 1032.048,A -85,B 0,C 180,E1 28909.337,E2 28909.337} C_VEL
LIN {X 0,Y 179.699,Z 1066.746,A -85,B 0,C 180,E1 28916.926,E2 28916.926} C_VEL
LIN {X 0,Y 188.084,Z 1102.187,A -85,B 0,C 180,E1 28924.303,E2 28924.303} C_VEL
LIN {X 0,Y 190.444,Z 1116.3,A -85,B 0,C 180,E1 28927.239,E2 28927.239} C_VEL
LIN {X 0,Y 176.498,Z 1155.219,A -85,B 0,C 180,E1 28934.059,E2 28934.059} C_VEL
LIN {X 0,Y 163.666,Z 1188.908,A -85,B 0,C 180,E1 28942.973,E2 28942.973} C_VEL
LIN {X 0,Y 153.528,Z 1217.879,A -85,B 0,C 180,E1 28954.423,E2 28954.423} C_VEL
LIN {X 0,Y 148.199,Z 1240.146,A -85,B 0,C 180,E1 28967.282,E2 28967.282} C_VEL
LIN {X 0,Y 147.097,Z 1255.608,A -85,B 0,C 180,E1 28979.958,E2 28979.958} C_VEL
LIN {X 0,Y 148.599,Z 1265.745,A -85,B 0,C 180,E1 28991.723,E2 28991.723} C_VEL
LIN {X 0,Y 159.619,Z 1275.632,A -85,B 0,C 180,E1 29008.289,E2 29008.289} C_VEL
LIN {X 0,Y 183.318,Z 1280.885,A -85,B 0,C 180,E1 29022.295,E2 29022.295} C_VEL
LIN {X 0,Y 182.326,Z 1281.135,A -85,B 0,C 180,E1 29023.553,E2 29023.553} C_VEL
LIN {X 0,Y 161.111,Z 1281.351,A -85,B 0,C 180,E1 29035.676,E2 29035.676} C_VEL
LIN {X 0,Y 149.289,Z 1277.592,A -85,B 0,C 180,E1 29052.301,E2 29052.301} C_VEL
LIN {X 0,Y 148.64,Z 1269.926,A -85,B 0,C 180,E1 29067.106,E2 29067.106} C_VEL
LIN {X 0,Y 148.937,Z 1263.615,A -85,B 0,C 180,E1 29074.403,E2 29074.403} C_VEL
LIN {X 0,Y 149.999,Z 1248.723,A -85,B 0,C 180,E1 29086.499,E2 29086.499} C_VEL
LIN {X 0,Y 159.51,Z 1249.202,A -85,B 0,C 180,E1 29104.779,E2 29104.779} C_VEL
LIN {X 0,Y 182.117,Z 1244.469,A -85,B 0,C 180,E1 29118.522,E2 29118.522} C_VEL
LIN {X 0,Y 209.591,Z 1236.542,A -85,B 0,C 180,E1 29127.303,E2 29127.303} C_VEL
LIN {X 0,Y 183.789,Z 1236.431,A -85,B 0,C 180,E1 29135.695,E2 29135.695} C_VEL
LIN {X 0,Y 165.008,Z 1231.07,A -85,B 0,C 180,E1 29145.9,E2 29145.9} C_VEL
LIN {X 0,Y 152.89,Z 1219.661,A -85,B 0,C 180,E1 29158.621,E2 29158.621} C_VEL
LIN {X 0,Y 149.139,Z 1203.663,A -85,B 0,C 180,E1 29171.023,E2 29171.023} C_VEL
LIN {X 0,Y 150.745,Z 1183.067,A -85,B 0,C 180,E1 29182.186,E2 29182.186} C_VEL
LIN {X 0,Y 155.465,Z 1157.845,A -85,B 0,C 180,E1 29191.636,E2 29191.636} C_VEL
LIN {X 0,Y 161.571,Z 1129.277,A -85,B 0,C 180,E1 29198.886,E2 29198.886} C_VEL
LIN {X 0,Y 168.073,Z 1095.637,A -85,B 0,C 180,E1 29204.345,E2 29204.345} C_VEL
LIN {X 0,Y 170.706,Z 1073.716,A -85,B 0,C 180,E1 29207.057,E2 29207.057} C_VEL
LIN {X 0,Y 160.662,Z 1030.91,A -85,B 0,C 180,E1 29214.267,E2 29214.267} C_VEL
LIN {X 0,Y 148.613,Z 994.337,A -85,B 0,C 180,E1 29221.833,E2 29221.833} C_VEL
LIN {X 0,Y 142.472,Z 977.53,A -85,B 0,C 180,E1 29226.048,E2 29226.048} C_VEL
LIN {X 0,Y 143.655,Z 977.53,A -85,B 0,C 180,E1 29237.793,E2 29237.793} C_VEL
LIN {X 0,Y 144.668,Z 977.53,A -85,B 0,C 180,E1 29243.96,E2 29243.96} C_VEL
LIN {X 0,Y 145.316,Z 977.53,A -85,B 0,C 180,E1 29251.466,E2 29251.466} C_VEL
LIN {X 0,Y 145.031,Z 977.7,A -85,B 0,C 180,E1 29252.967,E2 29252.967} C_VEL
LIN {X 0,Y 147.234,Z 983.222,A -85,B 0,C 180,E1 29254.954,E2 29254.954} C_VEL
LIN {X 0,Y 155.053,Z 999.711,A -85,B 0,C 180,E1 29260.778,E2 29260.778} C_VEL
LIN {X 0,Y 157.593,Z 1010.815,A -85,B 0,C 180,E1 29263.185,E2 29263.185} C_VEL
LIN {X 0,Y 160.561,Z 1030.392,A -85,B 0,C 180,E1 29266.743,E2 29266.743} C_VEL
LIN {X 0,Y 171.603,Z 1064.588,A -85,B 0,C 180,E1 29274.772,E2 29274.772} C_VEL
LIN {X 0,Y 179.738,Z 1098.634,A -85,B 0,C 180,E1 29282.231,E2 29282.231} C_VEL
LIN {X 0,Y 183.03,Z 1117.38,A -85,B 0,C 180,E1 29286.328,E2 29286.328} C_VEL
LIN {X 0,Y 168.66,Z 1156.124,A -85,B 0,C 180,E1 29293.399,E2 29293.399} C_VEL
LIN {X 0,Y 155.484,Z 1189.712,A -85,B 0,C 180,E1 29302.73,E2 29302.73} C_VEL
LIN {X 0,Y 145.397,Z 1218.083,A -85,B 0,C 180,E1 29314.589,E2 29314.589} C_VEL
LIN {X 0,Y 140.17,Z 1240.397,A -85,B 0,C 180,E1 29328.262,E2 29328.262} C_VEL
LIN {X 0,Y 139.366,Z 1255.602,A -85,B 0,C 180,E1 29341.513,E2 29341.513} C_VEL
LIN {X 0,Y 141.942,Z 1266.607,A -85,B 0,C 180,E1 29355.163,E2 29355.163} C_VEL
LIN {X 0,Y 155.855,Z 1276.403,A -85,B 0,C 180,E1 29372.274,E2 29372.274} C_VEL
LIN {X 0,Y 172.961,Z 1280.452,A -85,B 0,C 180,E1 29382.083,E2 29382.083} C_VEL
LIN {X 0,Y 173.438,Z 1280.709,A -85,B 0,C 180,E1 29383.136,E2 29383.136} C_VEL
LIN {X 0,Y 148.846,Z 1279.332,A -85,B 0,C 180,E1 29399.434,E2 29399.434} C_VEL
LIN {X 0,Y 140.563,Z 1273.274,A -85,B 0,C 180,E1 29417.579,E2 29417.579} C_VEL
LIN {X 0,Y 141.438,Z 1265.572,A -85,B 0,C 180,E1 29430.029,E2 29430.029} C_VEL
LIN {X 0,Y 141.352,Z 1254.197,A -85,B 0,C 180,E1 29440.842,E2 29440.842} C_VEL
LIN {X 0,Y 142.46,Z 1246.575,A -85,B 0,C 180,E1 29446.98,E2 29446.98} C_VEL
LIN {X 0,Y 153.028,Z 1247.754,A -85,B 0,C 180,E1 29466.482,E2 29466.482} C_VEL
LIN {X 0,Y 176.898,Z 1243.704,A -85,B 0,C 180,E1 29480.472,E2 29480.472} C_VEL
LIN {X 0,Y 197.953,Z 1238.575,A -85,B 0,C 180,E1 29487.391,E2 29487.391} C_VEL
LIN {X 0,Y 171.895,Z 1236.349,A -85,B 0,C 180,E1 29496.672,E2 29496.672} C_VEL
LIN {X 0,Y 153.011,Z 1228.228,A -85,B 0,C 180,E1 29508.619,E2 29508.619} C_VEL
LIN {X 0,Y 143.182,Z 1214.611,A -85,B 0,C 180,E1 29522.065,E2 29522.065} C_VEL
LIN {X 0,Y 141.464,Z 1195.798,A -85,B 0,C 180,E1 29535.31,E2 29535.31} C_VEL
LIN {X 0,Y 144.392,Z 1173.456,A -85,B 0,C 180,E1 29546.242,E2 29546.242} C_VEL
LIN {X 0,Y 150.012,Z 1146.458,A -85,B 0,C 180,E1 29555.309,E2 29555.309} C_VEL
LIN {X 0,Y 156.725,Z 1115.576,A -85,B 0,C 180,E1 29562.171,E2 29562.171} C_VEL
LIN {X 0,Y 163.368,Z 1075.905,A -85,B 0,C 180,E1 29567.71,E2 29567.71} C_VEL
LIN {X 0,Y 153.568,Z 1032.874,A -85,B 0,C 180,E1 29575.402,E2 29575.402} C_VEL
LIN {X 0,Y 141.779,Z 996.658,A -85,B 0,C 180,E1 29583.382,E2 29583.382} C_VEL
LIN {X 0,Y 134.618,Z 977.53,A -85,B 0,C 180,E1 29588.51,E2 29588.51} C_VEL
LIN {X 0,Y 135.579,Z 977.53,A -85,B 0,C 180,E1 29597.053,E2 29597.053} C_VEL
LIN {X 0,Y 137.41,Z 977.886,A -85,B 0,C 180,E1 29608.729,E2 29608.729} C_VEL
LIN {X 0,Y 148.535,Z 1001.756,A -85,B 0,C 180,E1 29618.405,E2 29618.405} C_VEL
LIN {X 0,Y 160.393,Z 1029.974,A -85,B 0,C 180,E1 29626.635,E2 29626.635} C_VEL
LIN {X 0,Y 160.561,Z 1030.392,A -85,B 0,C 180,E1 29626.743,E2 29626.743} C_VEL
LIN {X 0,Y 162.435,Z 1041.864,A -85,B 0,C 180,E1 29628.9,E2 29628.9} C_VEL
LIN {X 0,Y 163.452,Z 1061.793,A -85,B 0,C 180,E1 29632.281,E2 29632.281} C_VEL
LIN {X 0,Y 172.138,Z 1098.116,A -85,B 0,C 180,E1 29640.703,E2 29640.703} C_VEL
LIN {X 0,Y 175.399,Z 1118.764,A -85,B 0,C 180,E1 29645.41,E2 29645.41} C_VEL
LIN {X 0,Y 160.958,Z 1156.629,A -85,B 0,C 180,E1 29652.603,E2 29652.603} C_VEL
LIN {X 0,Y 147.074,Z 1191.102,A -85,B 0,C 180,E1 29662.703,E2 29662.703} C_VEL
LIN {X 0,Y 136.929,Z 1219.389,A -85,B 0,C 180,E1 29675.436,E2 29675.436} C_VEL
LIN {X 0,Y 132.209,Z 1240.408,A -85,B 0,C 180,E1 29689.22,E2 29689.22} C_VEL
LIN {X 0,Y 131.735,Z 1255.527,A -85,B 0,C 180,E1 29703.249,E2 29703.249} C_VEL
LIN {X 0,Y 136.1,Z 1267.709,A -85,B 0,C 180,E1 29719.461,E2 29719.461} C_VEL
LIN {X 0,Y 152.904,Z 1277.119,A -85,B 0,C 180,E1 29736.428,E2 29736.428} C_VEL
LIN {X 0,Y 163.779,Z 1279.814,A -85,B 0,C 180,E1 29742.377,E2 29742.377} C_VEL
LIN {X 0,Y 161.867,Z 1279.885,A -85,B 0,C 180,E1 29743.935,E2 29743.935} C_VEL
LIN {X 0,Y 137.443,Z 1276.338,A -85,B 0,C 180,E1 29763.866,E2 29763.866} C_VEL
LIN {X 0,Y 132.854,Z 1269.713,A -85,B 0,C 180,E1 29780.18,E2 29780.18} C_VEL
LIN {X 0,Y 133.807,Z 1263.349,A -85,B 0,C 180,E1 29790.03,E2 29790.03} C_VEL
LIN {X 0,Y 133.779,Z 1250.473,A -85,B 0,C 180,E1 29802.292,E2 29802.292} C_VEL
LIN {X 0,Y 134.943,Z 1244.289,A -85,B 0,C 180,E1 29807.343,E2 29807.343} C_VEL
LIN {X 0,Y 141.084,Z 1246.29,A -85,B 0,C 180,E1 29822.514,E2 29822.514} C_VEL
LIN {X 0,Y 162.294,Z 1244.45,A -85,B 0,C 180,E1 29838.362,E2 29838.362} C_VEL
LIN {X 0,Y 182.546,Z 1240.79,A -85,B 0,C 180,E1 29846.145,E2 29846.145} C_VEL
LIN {X 0,Y 185.556,Z 1239.83,A -85,B 0,C 180,E1 29847.767,E2 29847.767} C_VEL
LIN {X 0,Y 160.041,Z 1235.438,A -85,B 0,C 180,E1 29857.79,E2 29857.79} C_VEL
LIN {X 0,Y 142.307,Z 1225.127,A -85,B 0,C 180,E1 29870.855,E2 29870.855} C_VEL
LIN {X 0,Y 134.352,Z 1209.862,A -85,B 0,C 180,E1 29884.898,E2 29884.898} C_VEL
LIN {X 0,Y 133.97,Z 1190.155,A -85,B 0,C 180,E1 29898.026,E2 29898.026} C_VEL
LIN {X 0,Y 137.549,Z 1167.429,A -85,B 0,C 180,E1 29908.708,E2 29908.708} C_VEL
LIN {X 0,Y 144.009,Z 1138.753,A -85,B 0,C 180,E1 29917.861,E2 29917.861} C_VEL
LIN {X 0,Y 151.13,Z 1105.609,A -85,B 0,C 180,E1 29924.625,E2 29924.625} C_VEL
LIN {X 0,Y 156.007,Z 1077.799,A -85,B 0,C 180,E1 29928.467,E2 29928.467} C_VEL
LIN {X 0,Y 146.658,Z 1035.573,A -85,B 0,C 180,E1 29936.455,E2 29936.455} C_VEL
LIN {X 0,Y 135.289,Z 999.513,A -85,B 0,C 180,E1 29944.913,E2 29944.913} C_VEL
LIN {X 0,Y 126.88,Z 977.53,A -85,B 0,C 180,E1 29951.579,E2 29951.579} C_VEL
LIN {X 0,Y 128.415,Z 977.981,A -85,B 0,C 180,E1 29962.553,E2 29962.553} C_VEL
LIN {X 0,Y 132.195,Z 983.803,A -85,B 0,C 180,E1 29966.562,E2 29966.562} C_VEL
LIN {X 0,Y 136.218,Z 990.283,A -85,B 0,C 180,E1 29970.364,E2 29970.364} C_VEL
LIN {X 0,Y 148.182,Z 1017.019,A -85,B 0,C 180,E1 29980.467,E2 29980.467} C_VEL
LIN {X 0,Y 158.985,Z 1046.832,A -85,B 0,C 180,E1 29988.62,E2 29988.62} C_VEL
LIN {X 0,Y 163.452,Z 1061.793,A -85,B 0,C 180,E1 29992.281,E2 29992.281} C_VEL
LIN {X 0,Y 164.342,Z 1073.316,A -85,B 0,C 180,E1 29994.459,E2 29994.459} C_VEL
LIN {X 0,Y 163.64,Z 1093.025,A -85,B 0,C 180,E1 29997.949,E2 29997.949} C_VEL
LIN {X 0,Y 168.114,Z 1119.317,A -85,B 0,C 180,E1 30004.302,E2 30004.302} C_VEL
LIN {X 0,Y 152.953,Z 1157.912,A -85,B 0,C 180,E1 30011.959,E2 30011.959} C_VEL
LIN {X 0,Y 139.156,Z 1191.021,A -85,B 0,C 180,E1 30022.178,E2 30022.178} C_VEL
LIN {X 0,Y 128.826,Z 1219.328,A -85,B 0,C 180,E1 30035.64,E2 30035.64} C_VEL
LIN {X 0,Y 124.298,Z 1240.352,A -85,B 0,C 180,E1 30050.301,E2 30050.301} C_VEL
LIN {X 0,Y 124.01,Z 1253.868,A -85,B 0,C 180,E1 30063.452,E2 30063.452} C_VEL
LIN {X 0,Y 129.722,Z 1267.61,A -85,B 0,C 180,E1 30082.256,E2 30082.256} C_VEL
LIN {X 0,Y 153.01,Z 1278.37,A -85,B 0,C 180,E1 30101.887,E2 30101.887} C_VEL
LIN {X 0,Y 153.634,Z 1278.701,A -85,B 0,C 180,E1 30103.237,E2 30103.237} C_VEL
LIN {X 0,Y 130.467,Z 1274.558,A -85,B 0,C 180,E1 30122.353,E2 30122.353} C_VEL
LIN {X 0,Y 125.326,Z 1267.603,A -85,B 0,C 180,E1 30139.584,E2 30139.584} C_VEL
LIN {X 0,Y 126.205,Z 1260.981,A -85,B 0,C 180,E1 30150.032,E2 30150.032} C_VEL
LIN {X 0,Y 126.225,Z 1247.513,A -85,B 0,C 180,E1 30163.041,E2 30163.041} C_VEL
LIN {X 0,Y 127.488,Z 1241.89,A -85,B 0,C 180,E1 30167.91,E2 30167.91} C_VEL
LIN {X 0,Y 134.472,Z 1244.408,A -85,B 0,C 180,E1 30184.328,E2 30184.328} C_VEL
LIN {X 0,Y 157.104,Z 1243.201,A -85,B 0,C 180,E1 30200.538,E2 30200.538} C_VEL
LIN {X 0,Y 172.807,Z 1240.97,A -85,B 0,C 180,E1 30206.615,E2 30206.615} C_VEL
LIN {X 0,Y 174.279,Z 1240.415,A -85,B 0,C 180,E1 30207.771,E2 30207.771} C_VEL
LIN {X 0,Y 148.282,Z 1233.743,A -85,B 0,C 180,E1 30219.091,E2 30219.091} C_VEL
LIN {X 0,Y 131.823,Z 1221.182,A -85,B 0,C 180,E1 30233.448,E2 30233.448} C_VEL
LIN {X 0,Y 125.82,Z 1203.467,A -85,B 0,C 180,E1 30248.707,E2 30248.707} C_VEL
LIN {X 0,Y 127.04,Z 1182.164,A -85,B 0,C 180,E1 30261.934,E2 30261.934} C_VEL
LIN {X 0,Y 132.083,Z 1156.165,A -85,B 0,C 180,E1 30273.071,E2 30273.071} C_VEL
LIN {X 0,Y 138.979,Z 1126.734,A -85,B 0,C 180,E1 30281.428,E2 30281.428} C_VEL
LIN {X 0,Y 146.536,Z 1090.607,A -85,B 0,C 180,E1 30287.76,E2 30287.76} C_VEL
LIN {X 0,Y 148.31,Z 1077.788,A -85,B 0,C 180,E1 30289.617,E2 30289.617} C_VEL
LIN {X 0,Y 138.919,Z 1034.998,A -85,B 0,C 180,E1 30298.303,E2 30298.303} C_VEL
LIN {X 0,Y 127.861,Z 999.619,A -85,B 0,C 180,E1 30307.316,E2 30307.316} C_VEL
LIN {X 0,Y 119.437,Z 979.165,A -85,B 0,C 180,E1 30314.609,E2 30314.609} C_VEL
LIN {X 0,Y 124.111,Z 984.4,A -85,B 0,C 180,E1 30320.61,E2 30320.61} C_VEL
LIN {X 0,Y 130.946,Z 994.176,A -85,B 0,C 180,E1 30327.892,E2 30327.892} C_VEL
LIN {X 0,Y 140.966,Z 1016.885,A -85,B 0,C 180,E1 30337.348,E2 30337.348} C_VEL
LIN {X 0,Y 151.531,Z 1045.951,A -85,B 0,C 180,E1 30346.12,E2 30346.12} C_VEL
LIN {X 0,Y 160.384,Z 1078.305,A -85,B 0,C 180,E1 30354.387,E2 30354.387} C_VEL
LIN {X 0,Y 163.64,Z 1093.025,A -85,B 0,C 180,E1 30357.949,E2 30357.949} C_VEL
LIN {X 0,Y 163.671,Z 1108.265,A -85,B 0,C 180,E1 30361.069,E2 30361.069} C_VEL
LIN {X 0,Y 159.375,Z 1123.8,A -85,B 0,C 180,E1 30363.797,E2 30363.797} C_VEL
LIN {X 0,Y 143.857,Z 1161.529,A -85,B 0,C 180,E1 30371.878,E2 30371.878} C_VEL
LIN {X 0,Y 129.694,Z 1194.606,A -85,B 0,C 180,E1 30383.163,E2 30383.163} C_VEL
LIN {X 0,Y 120.32,Z 1220.58,A -85,B 0,C 180,E1 30396.771,E2 30396.771} C_VEL
LIN {X 0,Y 116.512,Z 1239.318,A -85,B 0,C 180,E1 30410.774,E2 30410.774} C_VEL
LIN {X 0,Y 116.481,Z 1253.652,A -85,B 0,C 180,E1 30425.545,E2 30425.545} C_VEL
LIN {X 0,Y 123.696,Z 1267.357,A -85,B 0,C 180,E1 30445.329,E2 30445.329} C_VEL
LIN {X 0,Y 144.662,Z 1277.112,A -85,B 0,C 180,E1 30462.884,E2 30462.884} C_VEL
LIN {X 0,Y 121.575,Z 1271.569,A -85,B 0,C 180,E1 30484.174,E2 30484.174} C_VEL
LIN {X 0,Y 118.065,Z 1262.277,A -85,B 0,C 180,E1 30504.511,E2 30504.511} C_VEL
LIN {X 0,Y 118.508,Z 1256.941,A -85,B 0,C 180,E1 30511.866,E2 30511.866} C_VEL
LIN {X 0,Y 120.117,Z 1239.332,A -85,B 0,C 180,E1 30528.637,E2 30528.637} C_VEL
LIN {X 0,Y 128.047,Z 1242.42,A -85,B 0,C 180,E1 30546.315,E2 30546.315} C_VEL
LIN {X 0,Y 155.458,Z 1241.536,A -85,B 0,C 180,E1 30564.263,E2 30564.263} C_VEL
LIN {X 0,Y 162.689,Z 1240.74,A -85,B 0,C 180,E1 30567.001,E2 30567.001} C_VEL
LIN {X 0,Y 155.078,Z 1238.578,A -85,B 0,C 180,E1 30570.804,E2 30570.804} C_VEL
LIN {X 0,Y 132.833,Z 1228.826,A -85,B 0,C 180,E1 30583.481,E2 30583.481} C_VEL
LIN {X 0,Y 120.475,Z 1213.475,A -85,B 0,C 180,E1 30599.117,E2 30599.117} C_VEL
LIN {X 0,Y 117.889,Z 1194.569,A -85,B 0,C 180,E1 30613.998,E2 30613.998} C_VEL
LIN {X 0,Y 120.827,Z 1171.688,A -85,B 0,C 180,E1 30626.885,E2 30626.885} C_VEL
LIN {X 0,Y 126.956,Z 1144.398,A -85,B 0,C 180,E1 30637.361,E2 30637.361} C_VEL
LIN {X 0,Y 134.602,Z 1112.052,A -85,B 0,C 180,E1 30645.323,E2 30645.323} C_VEL
LIN {X 0,Y 140.738,Z 1078.339,A -85,B 0,C 180,E1 30650.744,E2 30650.744} C_VEL
LIN {X 0,Y 132.286,Z 1038.34,A -85,B 0,C 180,E1 30659.415,E2 30659.415} C_VEL
LIN {X 0,Y 121.688,Z 1003.094,A -85,B 0,C 180,E1 30668.987,E2 30668.987} C_VEL
LIN {X 0,Y 116.532,Z 988.56,A -85,B 0,C 180,E1 30674.408,E2 30674.408} C_VEL
LIN {X 0,Y 118.873,Z 989.996,A -85,B 0,C 180,E1 30677.301,E2 30677.301} C_VEL
LIN {X 0,Y 122.247,Z 993.58,A -85,B 0,C 180,E1 30681.366,E2 30681.366} C_VEL
LIN {X 0,Y 127.628,Z 1001.454,A -85,B 0,C 180,E1 30687.211,E2 30687.211} C_VEL
LIN {X 0,Y 138.321,Z 1027.627,A -85,B 0,C 180,E1 30697.918,E2 30697.918} C_VEL
LIN {X 0,Y 147.894,Z 1057.982,A -85,B 0,C 180,E1 30707.023,E2 30707.023} C_VEL
LIN {X 0,Y 155.345,Z 1089.104,A -85,B 0,C 180,E1 30715.232,E2 30715.232} C_VEL
LIN {X 0,Y 160.9,Z 1119.16,A -85,B 0,C 180,E1 30722.966,E2 30722.966} C_VEL
LIN {X 0,Y 159.375,Z 1123.8,A -85,B 0,C 180,E1 30723.797,E2 30723.797} C_VEL
LIN {X 0,Y 152.872,Z 1134.499,A -85,B 0,C 180,E1 30725.324,E2 30725.324} C_VEL
LIN {X 0,Y 141.604,Z 1149.585,A -85,B 0,C 180,E1 30727.737,E2 30727.737} C_VEL
LIN {X 0,Y 140.763,Z 1151.348,A -85,B 0,C 180,E1 30728.144,E2 30728.144} C_VEL
LIN {X 0,Y 125.152,Z 1186.717,A -85,B 0,C 180,E1 30739.341,E2 30739.341} C_VEL
LIN {X 0,Y 113.639,Z 1216.047,A -85,B 0,C 180,E1 30754.262,E2 30754.262} C_VEL
LIN {X 0,Y 108.852,Z 1236.904,A -85,B 0,C 180,E1 30770.161,E2 30770.161} C_VEL
LIN {X 0,Y 108.855,Z 1251.749,A -85,B 0,C 180,E1 30785.935,E2 30785.935} C_VEL
LIN {X 0,Y 116.699,Z 1265.986,A -85,B 0,C 180,E1 30806.967,E2 30806.967} C_VEL
LIN {X 0,Y 134.587,Z 1274.934,A -85,B 0,C 180,E1 30822.426,E2 30822.426} C_VEL
LIN {X 0,Y 120.056,Z 1272.035,A -85,B 0,C 180,E1 30834.855,E2 30834.855} C_VEL
LIN {X 0,Y 110.441,Z 1263.033,A -85,B 0,C 180,E1 30858.161,E2 30858.161} C_VEL
LIN {X 0,Y 111.063,Z 1255.903,A -85,B 0,C 180,E1 30870.036,E2 30870.036} C_VEL
LIN {X 0,Y 111.519,Z 1240.139,A -85,B 0,C 180,E1 30885.806,E2 30885.806} C_VEL
LIN {X 0,Y 112.801,Z 1236.672,A -85,B 0,C 180,E1 30889.437,E2 30889.437} C_VEL
LIN {X 0,Y 121.809,Z 1240.284,A -85,B 0,C 180,E1 30908.503,E2 30908.503} C_VEL
LIN {X 0,Y 152.253,Z 1239.804,A -85,B 0,C 180,E1 30927.597,E2 30927.597} C_VEL
LIN {X 0,Y 129.067,Z 1230.554,A -85,B 0,C 180,E1 30939.432,E2 30939.432} C_VEL
LIN {X 0,Y 114.065,Z 1215.165,A -85,B 0,C 180,E1 30955.704,E2 30955.704} C_VEL
LIN {X 0,Y 110.05,Z 1194.994,A -85,B 0,C 180,E1 30972.722,E2 30972.722} C_VEL
LIN {X 0,Y 112.796,Z 1172.01,A -85,B 0,C 180,E1 30986.621,E2 30986.621} C_VEL
LIN {X 0,Y 119.39,Z 1143.213,A -85,B 0,C 180,E1 30998.283,E2 30998.283} C_VEL
LIN {X 0,Y 127.052,Z 1111.857,A -85,B 0,C 180,E1 31006.333,E2 31006.333} C_VEL
LIN {X 0,Y 133.342,Z 1079.792,A -85,B 0,C 180,E1 31011.802,E2 31011.802} C_VEL
LIN {X 0,Y 125.178,Z 1040.049,A -85,B 0,C 180,E1 31021.004,E2 31021.004} C_VEL
LIN {X 0,Y 115.511,Z 1006.384,A -85,B 0,C 180,E1 31030.819,E2 31030.819} C_VEL
LIN {X 0,Y 113.129,Z 998.89,A -85,B 0,C 180,E1 31033.926,E2 31033.926} C_VEL
LIN {X 0,Y 115.895,Z 997.049,A -85,B 0,C 180,E1 31036.38,E2 31036.38} C_VEL
LIN {X 0,Y 119.472,Z 1001.366,A -85,B 0,C 180,E1 31041.014,E2 31041.014} C_VEL
LIN {X 0,Y 123.586,Z 1007.598,A -85,B 0,C 180,E1 31045.762,E2 31045.762} C_VEL
LIN {X 0,Y 132.728,Z 1031.166,A -85,B 0,C 180,E1 31055.908,E2 31055.908} C_VEL
LIN {X 0,Y 141.711,Z 1061.049,A -85,B 0,C 180,E1 31065.47,E2 31065.47} C_VEL
LIN {X 0,Y 148.817,Z 1092.983,A -85,B 0,C 180,E1 31074.401,E2 31074.401} C_VEL
LIN {X 0,Y 153.477,Z 1120.8,A -85,B 0,C 180,E1 31081.945,E2 31081.945} C_VEL
LIN {X 0,Y 140.763,Z 1151.348,A -85,B 0,C 180,E1 31088.144,E2 31088.144} C_VEL
LIN {X 0,Y 131.234,Z 1164.365,A -85,B 0,C 180,E1 31091.056,E2 31091.056} C_VEL
LIN {X 0,Y 121.693,Z 1176.766,A -85,B 0,C 180,E1 31094.715,E2 31094.715} C_VEL
LIN {X 0,Y 108.915,Z 1206.305,A -85,B 0,C 180,E1 31108.49,E2 31108.49} C_VEL
LIN {X 0,Y 101.912,Z 1230.162,A -85,B 0,C 180,E1 31125.623,E2 31125.623} C_VEL
LIN {X 0,Y 100.889,Z 1246.298,A -85,B 0,C 180,E1 31142.09,E2 31142.09} C_VEL
LIN {X 0,Y 104.723,Z 1259.251,A -85,B 0,C 180,E1 31160.202,E2 31160.202} C_VEL
LIN {X 0,Y 122.861,Z 1271.68,A -85,B 0,C 180,E1 31181.001,E2 31181.001} C_VEL
LIN {X 0,Y 124.797,Z 1272.611,A -85,B 0,C 180,E1 31183.286,E2 31183.286} C_VEL
LIN {X 0,Y 104.464,Z 1264.351,A -85,B 0,C 180,E1 31208.78,E2 31208.78} C_VEL
LIN {X 0,Y 103.645,Z 1254.693,A -85,B 0,C 180,E1 31227.944,E2 31227.944} C_VEL
LIN {X 0,Y 103.339,Z 1241.357,A -85,B 0,C 180,E1 31242.746,E2 31242.746} C_VEL
LIN {X 0,Y 105.565,Z 1233.803,A -85,B 0,C 180,E1 31250.092,E2 31250.092} C_VEL
LIN {X 0,Y 115.815,Z 1238.009,A -85,B 0,C 180,E1 31270.903,E2 31270.903} C_VEL
LIN {X 0,Y 141.209,Z 1238.547,A -85,B 0,C 180,E1 31287.608,E2 31287.608} C_VEL
LIN {X 0,Y 117.548,Z 1226.812,A -85,B 0,C 180,E1 31301.258,E2 31301.258} C_VEL
LIN {X 0,Y 104.798,Z 1210.197,A -85,B 0,C 180,E1 31318.379,E2 31318.379} C_VEL
LIN {X 0,Y 102.442,Z 1188.995,A -85,B 0,C 180,E1 31335.903,E2 31335.903} C_VEL
LIN {X 0,Y 106.35,Z 1164.291,A -85,B 0,C 180,E1 31350.304,E2 31350.304} C_VEL
LIN {X 0,Y 113.536,Z 1135.782,A -85,B 0,C 180,E1 31361.287,E2 31361.287} C_VEL
LIN {X 0,Y 121.694,Z 1102.483,A -85,B 0,C 180,E1 31369.255,E2 31369.255} C_VEL
LIN {X 0,Y 125.892,Z 1080.988,A -85,B 0,C 180,E1 31372.96,E2 31372.96} C_VEL
LIN {X 0,Y 118.257,Z 1042.029,A -85,B 0,C 180,E1 31382.697,E2 31382.697} C_VEL
LIN {X 0,Y 109.465,Z 1009.329,A -85,B 0,C 180,E1 31393.114,E2 31393.114} C_VEL
LIN {X 0,Y 114.197,Z 1005.301,A -85,B 0,C 180,E1 31397.128,E2 31397.128} C_VEL
LIN {X 0,Y 119.575,Z 1013.498,A -85,B 0,C 180,E1 31404.112,E2 31404.112} C_VEL
LIN {X 0,Y 128.057,Z 1036.93,A -85,B 0,C 180,E1 31414.618,E2 31414.618} C_VEL
LIN {X 0,Y 135.751,Z 1065.208,A -85,B 0,C 180,E1 31424.178,E2 31424.178} C_VEL
LIN {X 0,Y 142.121,Z 1096.05,A -85,B 0,C 180,E1 31433.267,E2 31433.267} C_VEL
LIN {X 0,Y 146.075,Z 1121.156,A -85,B 0,C 180,E1 31440.501,E2 31440.501} C_VEL
LIN {X 0,Y 130.24,Z 1158.297,A -85,B 0,C 180,E1 31448.787,E2 31448.787} C_VEL
LIN {X 0,Y 121.693,Z 1176.766,A -85,B 0,C 180,E1 31454.715,E2 31454.715} C_VEL
LIN {X 0,Y 115.065,Z 1185.876,A -85,B 0,C 180,E1 31458.056,E2 31458.056} C_VEL
LIN {X 0,Y 104.071,Z 1198.308,A -85,B 0,C 180,E1 31463.758,E2 31463.758} C_VEL
LIN {X 0,Y 103.365,Z 1199.772,A -85,B 0,C 180,E1 31464.568,E2 31464.568} C_VEL
LIN {X 0,Y 95.084,Z 1223.723,A -85,B 0,C 180,E1 31481.348,E2 31481.348} C_VEL
LIN {X 0,Y 93.064,Z 1241.129,A -85,B 0,C 180,E1 31498.767,E2 31498.767} C_VEL
LIN {X 0,Y 95.429,Z 1253.802,A -85,B 0,C 180,E1 31516.064,E2 31516.064} C_VEL
LIN {X 0,Y 110.065,Z 1267.176,A -85,B 0,C 180,E1 31538.204,E2 31538.204} C_VEL
LIN {X 0,Y 115.303,Z 1269.668,A -85,B 0,C 180,E1 31542.294,E2 31542.294} C_VEL
LIN {X 0,Y 113.649,Z 1269.456,A -85,B 0,C 180,E1 31544.817,E2 31544.817} C_VEL
LIN {X 0,Y 96.344,Z 1260.04,A -85,B 0,C 180,E1 31571.71,E2 31571.71} C_VEL
LIN {X 0,Y 96.205,Z 1251.827,A -85,B 0,C 180,E1 31587.785,E2 31587.785} C_VEL
LIN {X 0,Y 96.093,Z 1236.851,A -85,B 0,C 180,E1 31604.891,E2 31604.891} C_VEL
LIN {X 0,Y 98.453,Z 1230.843,A -85,B 0,C 180,E1 31611.243,E2 31611.243} C_VEL
LIN {X 0,Y 110.078,Z 1235.607,A -85,B 0,C 180,E1 31633.544,E2 31633.544} C_VEL
LIN {X 0,Y 128.079,Z 1236.848,A -85,B 0,C 180,E1 31645.965,E2 31645.965} C_VEL
LIN {X 0,Y 129.488,Z 1236.357,A -85,B 0,C 180,E1 31647.859,E2 31647.859} C_VEL
LIN {X 0,Y 108.076,Z 1223.937,A -85,B 0,C 180,E1 31661.674,E2 31661.674} C_VEL
LIN {X 0,Y 95.89,Z 1204.844,A -85,B 0,C 180,E1 31681.196,E2 31681.196} C_VEL
LIN {X 0,Y 95.004,Z 1183.603,A -85,B 0,C 180,E1 31698.668,E2 31698.668} C_VEL
LIN {X 0,Y 99.874,Z 1157.759,A -85,B 0,C 180,E1 31713.485,E2 31713.485} C_VEL
LIN {X 0,Y 107.506,Z 1129.051,A -85,B 0,C 180,E1 31724.175,E2 31724.175} C_VEL
LIN {X 0,Y 116.605,Z 1092.478,A -85,B 0,C 180,E1 31732.405,E2 31732.405} C_VEL
LIN {X 0,Y 118.239,Z 1080.48,A -85,B 0,C 180,E1 31734.686,E2 31734.686} C_VEL
LIN {X 0,Y 111.201,Z 1043.211,A -85,B 0,C 180,E1 31744.757,E2 31744.757} C_VEL
LIN {X 0,Y 105.97,Z 1020.3,A -85,B 0,C 180,E1 31752.674,E2 31752.674} C_VEL
LIN {X 0,Y 112.379,Z 1013.982,A -85,B 0,C 180,E1 31757.887,E2 31757.887} C_VEL
LIN {X 0,Y 116.067,Z 1020.746,A -85,B 0,C 180,E1 31763.107,E2 31763.107} C_VEL
LIN {X 0,Y 123.063,Z 1042.068,A -85,B 0,C 180,E1 31773.048,E2 31773.048} C_VEL
LIN {X 0,Y 130.338,Z 1071.26,A -85,B 0,C 180,E1 31783.413,E2 31783.413} C_VEL
LIN {X 0,Y 136.313,Z 1104.336,A -85,B 0,C 180,E1 31793.731,E2 31793.731} C_VEL
LIN {X 0,Y 138.573,Z 1123.123,A -85,B 0,C 180,E1 31799.368,E2 31799.368} C_VEL
LIN {X 0,Y 121.782,Z 1160.258,A -85,B 0,C 180,E1 31808.093,E2 31808.093} C_VEL
LIN {X 0,Y 106.356,Z 1193.07,A -85,B 0,C 180,E1 31820.954,E2 31820.954} C_VEL
LIN {X 0,Y 103.365,Z 1199.772,A -85,B 0,C 180,E1 31824.568,E2 31824.568} C_VEL
LIN {X 0,Y 97.573,Z 1207.865,A -85,B 0,C 180,E1 31829.466,E2 31829.466} C_VEL
LIN {X 0,Y 87.891,Z 1219.976,A -85,B 0,C 180,E1 31839.229,E2 31839.229} C_VEL
LIN {X 0,Y 85.444,Z 1238.515,A -85,B 0,C 180,E1 31858.657,E2 31858.657} C_VEL
LIN {X 0,Y 87.41,Z 1249.926,A -85,B 0,C 180,E1 31874.625,E2 31874.625} C_VEL
LIN {X 0,Y 105.334,Z 1266.224,A -85,B 0,C 180,E1 31901.853,E2 31901.853} C_VEL
LIN {X 0,Y 106.269,Z 1266.658,A -85,B 0,C 180,E1 31902.587,E2 31902.587} C_VEL
LIN {X 0,Y 105.537,Z 1266.615,A -85,B 0,C 180,E1 31904.175,E2 31904.175} C_VEL
LIN {X 0,Y 88.857,Z 1256.296,A -85,B 0,C 180,E1 31932.762,E2 31932.762} C_VEL
LIN {X 0,Y 88.752,Z 1248.934,A -85,B 0,C 180,E1 31947.599,E2 31947.599} C_VEL
LIN {X 0,Y 89.23,Z 1232.09,A -85,B 0,C 180,E1 31967.335,E2 31967.335} C_VEL
LIN {X 0,Y 91.377,Z 1227.634,A -85,B 0,C 180,E1 31972.079,E2 31972.079} C_VEL
LIN {X 0,Y 104.633,Z 1233.084,A -85,B 0,C 180,E1 31996.449,E2 31996.449} C_VEL
LIN {X 0,Y 116.404,Z 1234.31,A -85,B 0,C 180,E1 32005.043,E2 32005.043} C_VEL
LIN {X 0,Y 118.909,Z 1233.978,A -85,B 0,C 180,E1 32007.668,E2 32007.668} C_VEL
LIN {X 0,Y 96.864,Z 1218.679,A -85,B 0,C 180,E1 32024.18,E2 32024.18} C_VEL
LIN {X 0,Y 87.245,Z 1198.288,A -85,B 0,C 180,E1 32045.053,E2 32045.053} C_VEL
LIN {X 0,Y 88.048,Z 1176.222,A -85,B 0,C 180,E1 32062.855,E2 32062.855} C_VEL
LIN {X 0,Y 93.933,Z 1150.121,A -85,B 0,C 180,E1 32077.312,E2 32077.312} C_VEL
LIN {X 0,Y 102.597,Z 1118.583,A -85,B 0,C 180,E1 32088.247,E2 32088.247} C_VEL
LIN {X 0,Y 111.113,Z 1083.293,A -85,B 0,C 180,E1 32095.689,E2 32095.689} C_VEL
LIN {X 0,Y 104.653,Z 1046.16,A -85,B 0,C 180,E1 32106.494,E2 32106.494} C_VEL
LIN {X 0,Y 101.769,Z 1031.752,A -85,B 0,C 180,E1 32111.678,E2 32111.678} C_VEL
LIN {X 0,Y 110.316,Z 1022.822,A -85,B 0,C 180,E1 32118.459,E2 32118.459} C_VEL
LIN {X 0,Y 113.532,Z 1030.989,A -85,B 0,C 180,E1 32123.764,E2 32123.764} C_VEL
LIN {X 0,Y 120.049,Z 1054.83,A -85,B 0,C 180,E1 32134.488,E2 32134.488} C_VEL
LIN {X 0,Y 126.335,Z 1085.928,A -85,B 0,C 180,E1 32145.539,E2 32145.539} C_VEL
LIN {X 0,Y 130.908,Z 1118.562,A -85,B 0,C 180,E1 32156.152,E2 32156.152} C_VEL
LIN {X 0,Y 131.054,Z 1124.507,A -85,B 0,C 180,E1 32157.966,E2 32157.966} C_VEL
LIN {X 0,Y 113.305,Z 1162.25,A -85,B 0,C 180,E1 32167.354,E2 32167.354} C_VEL
LIN {X 0,Y 97.436,Z 1194.955,A -85,B 0,C 180,E1 32181.458,E2 32181.458} C_VEL
